C01818=1037.554,349.984,372.996,172.475,44.077,158.586
C01819=1037.561,350.231,372.958,172.480,44.080,158.587
C01820=1037.569,350.478,372.921,172.487,44.083,158.588
C01821=1037.577,350.725,372.883,172.492,44.085,158.589
C01822=1037.584,350.973,372.845,172.498,44.089,158.591
C01823=1037.592,351.220,372.808,172.503,44.092,158.592
C01824=1037.599,351.466,372.769,172.510,44.094,158.593
C01825=1037.607,351.714,372.731,172.515,44.097,158.594
C01826=1037.615,351.960,372.694,172.521,44.100,158.595
C01827=1037.623,352.207,372.656,172.526,44.102,158.596
C01828=1037.631,352.455,372.618,172.533,44.105,158.598
C01829=1037.638,352.702,372.580,172.538,44.108,158.599
C01830=1037.645,352.948,372.542,172.544,44.111,158.600
C01831=1037.653,353.196,372.504,172.550,44.114,158.601
C01832=1037.661,353.443,372.466,172.556,44.116,158.602
C01833=1037.668,353.689,372.427,172.561,44.119,158.604
C01834=1037.677,353.937,372.390,172.568,44.122,158.605
C01835=1037.685,354.183,372.352,172.574,44.125,158.606
C01836=1037.692,354.431,372.314,172.579,44.128,158.607
C01837=1037.700,354.678,372.276,172.586,44.130,158.608
C01838=1037.708,354.924,372.238,172.591,44.134,158.610
C01839=1037.716,355.171,372.199,172.598,44.136,158.611
C01840=1037.723,355.418,372.161,172.603,44.139,158.612
C01841=1037.731,355.666,372.123,172.609,44.142,158.613
C01842=1037.739,355.912,372.085,172.616,44.145,158.615
C01843=1037.747,356.159,372.047,172.621,44.148,158.616
C01844=1037.754,356.406,372.008,172.628,44.151,158.617
C01845=1037.762,356.653,371.969,172.633,44.154,158.619
C01846=1037.770,356.900,371.931,172.639,44.157,158.620
C01847=1037.778,357.147,371.892,172.646,44.160,158.621
C01848=1037.786,357.393,371.854,172.651,44.163,158.622
C01849=1037.794,357.641,371.815,172.658,44.166,158.624
C01850=1037.801,357.887,371.777,172.663,44.168,158.625
C01851=1037.810,358.134,371.739,172.670,44.172,158.626
C01852=1037.818,358.381,371.700,172.676,44.175,158.627
C01853=1037.825,358.628,371.662,172.681,44.178,158.629
C01854=1037.833,358.875,371.623,172.688,44.181,158.630
C01855=1037.841,359.122,371.585,172.694,44.184,158.631
C01856=1037.848,359.369,371.546,172.700,44.187,158.632
C01857=1037.857,359.616,371.506,172.706,44.190,158.634
C01858=1037.864,359.862,371.468,172.713,44.193,158.635
C01859=1037.873,360.110,371.429,172.718,44.196,158.636
C01860=1037.881,360.356,371.390,172.725,44.199,158.638
C01861=1037.889,360.603,371.352,172.731,44.202,158.639
C01862=1037.897,360.850,371.313,172.737,44.205,158.640
C01863=1037.904,361.097,371.273,172.744,44.208,158.642
C01864=1037.912,361.343,371.235,172.750,44.212,158.643
C01865=1037.920,361.591,371.196,172.757,44.215,158.644
C01866=1037.929,361.837,371.157,172.762,44.218,158.646
C01867=1037.937,362.084,371.119,172.769,44.221,158.647
C01868=1037.944,362.331,371.079,172.775,44.225,158.648
C01869=1037.952,362.578,371.040,172.782,44.228,158.650
C01870=1037.964,362.950,370.981,172.791,44.233,158.652
C01871=1037.975,363.322,370.922,172.801,44.237,158.654
C01872=1037.988,363.694,370.862,172.811,44.242,158.656
C01873=1037.999,364.067,370.803,172.819,44.248,158.658
C01874=1038.008,364.313,370.764,172.826,44.251,158.659
C01875=1038.016,364.560,370.724,172.833,44.254,158.661
C01876=1038.023,364.806,370.685,172.839,44.258,158.662
C01877=1038.031,365.053,370.645,172.846,44.261,158.664
C01878=1038.039,365.300,370.607,172.852,44.264,158.665
C01879=1038.048,365.547,370.567,172.858,44.267,158.666
C01880=1038.056,365.794,370.527,172.865,44.271,158.668
C01881=1038.064,366.040,370.488,172.872,44.274,158.669
C01882=1038.072,366.287,370.448,172.877,44.277,158.671
C01883=1038.080,366.534,370.409,172.884,44.281,158.672
C01884=1038.088,366.781,370.369,172.891,44.284,158.674
C01885=1038.096,367.027,370.330,172.897,44.288,158.675
C01886=1038.104,367.274,370.290,172.904,44.291,158.676
C01887=1038.113,367.521,370.250,172.911,44.295,158.678
C01888=1038.121,367.767,370.211,172.917,44.298,158.679
C01889=1038.129,368.014,370.171,172.924,44.302,158.681
C01890=1038.137,368.260,370.131,172.931,44.305,158.682
C01891=1038.145,368.507,370.091,172.938,44.308,158.684
C01892=1038.154,368.754,370.052,172.943,44.312,158.685
C01893=1038.161,369.001,370.012,172.950,44.315,158.687
C01894=1038.170,369.247,369.973,172.957,44.318,158.688
C01895=1038.178,369.493,369.932,172.964,44.322,158.690
C01896=1038.186,369.740,369.893,172.971,44.326,158.691
C01897=1038.195,369.988,369.852,172.977,44.329,158.692
C01898=1038.203,370.234,369.812,172.984,44.333,158.694
C01899=1038.211,370.480,369.772,172.991,44.336,158.696
C01900=1038.219,370.727,369.732,172.998,44.340,158.697
C01901=1038.228,370.973,369.692,173.005,44.343,158.699
C01902=1038.236,371.220,369.652,173.011,44.347,158.700
C01903=1038.243,371.467,369.612,173.018,44.351,158.702
C01904=1038.251,371.713,369.571,173.025,44.355,158.703
C01905=1038.260,371.960,369.530,173.032,44.358,158.705
C01906=1038.268,372.206,369.491,173.039,44.362,158.706
C01907=1038.276,372.453,369.450,173.046,44.366,158.708
C01908=1038.285,372.699,369.410,173.053,44.369,158.709
C01909=1038.293,372.947,369.369,173.059,44.373,158.711
C01910=1038.302,373.193,369.329,173.066,44.377,158.712
C01911=1038.310,373.439,369.289,173.073,44.380,158.714
C01912=1038.318,373.685,369.248,173.080,44.384,158.716
C01913=1038.326,373.932,369.207,173.087,44.388,158.717
C01914=1038.334,374.179,369.167,173.094,44.391,158.719
C01915=1038.343,374.425,369.127,173.101,44.395,158.720
C01916=1038.351,374.672,369.086,173.108,44.399,158.722
C01917=1038.359,374.918,369.045,173.115,44.403,158.724
C01918=1038.367,375.165,369.005,173.122,44.406,158.725
C01919=1038.376,375.412,368.964,173.130,44.411,158.727
C01920=1038.384,375.658,368.923,173.137,44.414,158.728
C01921=1038.393,375.904,368.883,173.144,44.418,158.730
C01922=1038.401,376.151,368.842,173.151,44.422,158.732
C01923=1038.410,376.397,368.801,173.158,44.426,158.733
C01924=1038.418,376.643,368.760,173.165,44.429,158.735
C01925=1038.426,376.890,368.719,173.172,44.433,158.736
C01926=1038.441,377.283,368.654,173.184,44.439,158.739
C01927=1038.454,377.675,368.590,173.195,44.446,158.742
C01928=1038.468,378.068,368.524,173.207,44.452,158.744
C01929=1038.482,378.461,368.459,173.218,44.458,158.747
C01930=1038.489,378.707,368.417,173.225,44.462,158.749
C01931=1038.498,378.954,368.376,173.233,44.467,158.750
C01932=1038.506,379.200,368.335,173.240,44.470,158.752
C01933=1038.515,379.447,368.294,173.247,44.474,158.754
C01934=1038.523,379.692,368.252,173.254,44.478,158.755
C01935=1038.532,379.939,368.211,173.261,44.483,158.757
C01936=1038.541,380.184,368.169,173.270,44.487,158.759
C01937=1038.549,380.431,368.128,173.277,44.491,158.761
C01938=1038.558,380.677,368.087,173.284,44.495,158.762
C01939=1038.566,380.923,368.045,173.292,44.499,158.764
C01940=1038.574,381.169,368.003,173.299,44.503,158.766
C01941=1038.583,381.416,367.962,173.306,44.507,158.768
C01942=1038.591,381.662,367.921,173.315,44.511,158.769
C01943=1038.600,381.908,367.879,173.322,44.516,158.771
C01944=1038.609,382.155,367.838,173.329,44.520,158.773
C01945=1038.618,382.401,367.796,173.336,44.524,158.775
C01946=1038.625,382.647,367.754,173.344,44.528,158.776
C01947=1038.634,382.893,367.712,173.352,44.532,158.778
C01948=1038.643,383.140,367.670,173.360,44.537,158.780
C01949=1038.652,383.386,367.629,173.367,44.541,158.782
C01950=1038.661,383.633,367.587,173.374,44.545,158.783
C01951=1038.669,383.878,367.546,173.383,44.549,158.785
C01952=1038.678,384.125,367.503,173.390,44.554,158.787
C01953=1038.687,384.371,367.462,173.397,44.558,158.789
C01954=1038.696,384.618,367.420,173.406,44.562,158.791
C01955=1038.704,384.864,367.378,173.413,44.567,158.793
C01956=1038.714,385.110,367.336,173.421,44.571,158.794
C01957=1038.722,385.356,367.293,173.428,44.575,158.796
C01958=1038.731,385.603,367.252,173.436,44.579,158.798
C01959=1038.740,385.849,367.210,173.444,44.584,158.800
C01960=1038.749,386.095,367.168,173.452,44.588,158.802
C01961=1038.758,386.341,367.126,173.460,44.593,158.804
C01962=1038.766,386.588,367.084,173.467,44.597,158.805
C01963=1038.775,386.834,367.041,173.476,44.601,158.807
C01964=1038.784,387.080,366.999,173.483,44.606,158.809
C01965=1038.794,387.326,366.957,173.492,44.610,158.811
C01966=1038.802,387.572,366.915,173.499,44.615,158.813
C01967=1038.811,387.818,366.872,173.508,44.619,158.815
C01968=1038.820,388.065,366.831,173.515,44.624,158.817
C01969=1038.829,388.311,366.787,173.523,44.628,158.819
C01970=1038.838,388.557,366.745,173.531,44.632,158.821
C01971=1038.847,388.803,366.703,173.539,44.637,158.823
C01972=1038.856,389.050,366.660,173.548,44.642,158.825
C01973=1038.865,389.295,366.618,173.555,44.646,158.826
C01974=1038.873,389.541,366.574,173.564,44.651,158.828
C01975=1038.883,389.787,366.532,173.571,44.655,158.830
C01976=1038.892,390.034,366.489,173.580,44.660,158.832
C01977=1038.901,390.280,366.447,173.588,44.665,158.834
C01978=1038.909,390.526,366.404,173.596,44.670,158.836
C01979=1038.918,390.772,366.361,173.604,44.674,158.838
C01980=1038.928,391.019,366.318,173.613,44.679,158.840
C01981=1038.937,391.264,366.276,173.621,44.684,158.842
C01982=1038.945,391.477,366.238,173.627,44.687,158.844
C01983=1038.952,391.691,366.201,173.635,44.692,158.846
C01984=1038.959,391.904,366.163,173.642,44.696,158.847
C01985=1038.967,392.117,366.126,173.649,44.700,158.849
C01986=1038.976,392.331,366.088,173.657,44.704,158.851
C01987=1038.983,392.544,366.051,173.664,44.709,158.853
C01988=1038.991,392.757,366.014,173.672,44.713,158.855
C01989=1038.999,392.971,365.976,173.679,44.717,158.856
C01990=1039.009,393.217,365.933,173.687,44.721,158.858
C01991=1039.017,393.463,365.890,173.696,44.726,158.861
C01992=1039.026,393.709,365.846,173.704,44.731,158.863
C01993=1039.036,393.955,365.804,173.712,44.736,158.865
C01994=1039.045,394.201,365.760,173.721,44.741,158.867
C01995=1039.054,394.447,365.717,173.730,44.746,158.869
C01996=1039.064,394.693,365.673,173.737,44.751,158.871
C01997=1039.072,394.939,365.630,173.746,44.756,158.873
C01998=1039.082,395.185,365.586,173.755,44.761,158.875
C01999=1039.091,395.430,365.543,173.764,44.766,158.877
C02000=1039.100,395.677,365.499,173.772,44.771,158.879
C02001=1039.109,395.922,365.456,173.781,44.776,158.882
C02002=1039.119,396.168,365.412,173.790,44.781,158.884
C02003=1039.127,396.414,365.368,173.799,44.786,158.886
C02004=1039.136,396.660,365.324,173.807,44.791,158.888
C02005=1039.147,396.906,365.281,173.815,44.796,158.890
C02006=1039.155,397.152,365.237,173.824,44.801,158.892
C02007=1039.165,397.398,365.193,173.833,44.806,158.895
C02008=1039.174,397.644,365.149,173.842,44.811,158.897
C02009=1039.183,397.889,365.105,173.851,44.816,158.899
C02010=1039.192,398.136,365.061,173.860,44.821,158.901
C02011=1039.203,398.381,365.018,173.869,44.826,158.903
C02012=1039.212,398.627,364.973,173.878,44.832,158.906
C02013=1039.221,398.873,364.930,173.887,44.837,158.908
C02014=1039.231,399.118,364.885,173.896,44.842,158.910
C02015=1039.240,399.365,364.841,173.904,44.848,158.912
C02016=1039.249,399.611,364.797,173.913,44.853,158.914
C02017=1039.259,399.857,364.753,173.922,44.858,158.917
C02018=1039.268,400.102,364.708,173.931,44.863,158.919
C02019=1039.277,400.348,364.664,173.940,44.868,158.921
C02020=1039.287,400.594,364.620,173.949,44.874,158.924
C02021=1039.296,400.839,364.575,173.958,44.879,158.926
C02022=1039.306,401.086,364.531,173.968,44.884,158.928
C02023=1039.316,401.331,364.486,173.978,44.890,158.931
C02024=1039.325,401.577,364.442,173.987,44.895,158.933
C02025=1039.335,401.823,364.397,173.996,44.901,158.935
C02026=1039.344,402.068,364.352,174.005,44.906,158.938
C02027=1039.354,402.314,364.308,174.014,44.911,158.940
C02028=1039.363,402.560,364.263,174.023,44.917,158.942
C02029=1039.373,402.805,364.219,174.032,44.922,158.945
C02030=1039.382,403.051,364.173,174.042,44.928,158.947
C02031=1039.392,403.298,364.129,174.051,44.934,158.949
C02032=1039.402,403.544,364.084,174.061,44.939,158.952
C02033=1039.412,403.789,364.039,174.070,44.944,158.954
C02034=1039.421,404.035,363.994,174.080,44.950,158.957
C02035=1039.430,404.280,363.949,174.089,44.956,158.959
C02036=1039.440,404.526,363.904,174.098,44.961,158.961
C02037=1039.450,404.771,363.859,174.108,44.967,158.964
C02038=1039.459,405.018,363.813,174.118,44.973,158.966
C02039=1039.469,405.263,363.768,174.127,44.978,158.969
C02040=1039.479,405.508,363.723,174.137,44.984,158.971
C02041=1039.488,405.754,363.678,174.147,44.989,158.974
C02042=1039.498,405.978,363.637,174.155,44.995,158.976
C02043=1039.506,406.201,363.595,174.164,45.000,158.978
C02044=1039.515,406.424,363.554,174.173,45.005,158.981
C02045=1039.525,406.647,363.513,174.182,45.010,158.983
C02046=1039.533,406.870,363.471,174.190,45.016,158.985
C02047=1039.542,407.093,363.431,174.199,45.021,158.987
C02048=1039.551,407.317,363.389,174.208,45.026,158.990
C02049=1039.560,407.540,363.347,174.218,45.032,158.992
C02050=1039.570,407.786,363.302,174.227,45.038,158.995
C02051=1039.580,408.031,363.256,174.238,45.043,158.997
C02052=1039.590,408.277,363.211,174.247,45.049,159.000
C02053=1039.599,408.523,363.165,174.257,45.055,159.002
C02054=1039.609,408.769,363.120,174.267,45.061,159.005
C02055=1039.620,409.014,363.074,174.277,45.067,159.007
C02056=1039.629,409.260,363.028,174.287,45.073,159.010
C02057=1039.640,409.505,362.982,174.297,45.079,159.013
C02058=1039.650,409.750,362.936,174.307,45.084,159.015
C02059=1039.660,409.997,362.890,174.318,45.090,159.018
C02060=1039.670,410.242,362.844,174.327,45.097,159.020
C02061=1039.680,410.487,362.799,174.338,45.102,159.023
C02062=1039.690,410.733,362.752,174.348,45.109,159.026
C02063=1039.701,410.979,362.706,174.358,45.115,159.028
C02064=1039.711,411.223,362.661,174.369,45.120,159.031
C02065=1039.721,411.469,362.614,174.379,45.127,159.034
C02066=1039.731,411.715,362.569,174.389,45.133,159.037
C02067=1039.741,411.960,362.521,174.400,45.139,159.039
C02068=1039.751,412.206,362.475,174.410,45.145,159.042
C02069=1039.762,412.452,362.429,174.420,45.152,159.045
C02070=1039.772,412.696,362.382,174.431,45.158,159.047
C02071=1039.781,412.942,362.336,174.441,45.164,159.050
C02072=1039.792,413.188,362.290,174.452,45.170,159.053
C02073=1039.802,413.433,362.242,174.462,45.176,159.056
C02074=1039.812,413.679,362.196,174.473,45.183,159.058
C02075=1039.823,413.924,362.149,174.484,45.189,159.061
C02076=1039.833,414.169,362.102,174.494,45.196,159.064
C02077=1039.843,414.415,362.056,174.505,45.202,159.067
C02078=1039.854,414.660,362.009,174.516,45.208,159.070
C02079=1039.864,414.905,361.962,174.527,45.215,159.073
C02080=1039.874,415.151,361.915,174.538,45.221,159.075
C02081=1039.884,415.397,361.868,174.548,45.228,159.078
C02082=1039.895,415.642,361.821,174.559,45.234,159.081
C02083=1039.905,415.887,361.774,174.570,45.241,159.084
C02084=1039.916,416.132,361.727,174.581,45.247,159.087
C02085=1039.927,416.378,361.680,174.592,45.254,159.090
C02086=1039.937,416.623,361.633,174.603,45.260,159.093
C02087=1039.948,416.868,361.586,174.614,45.266,159.096
C02088=1039.959,417.113,361.539,174.625,45.273,159.099
C02089=1039.969,417.359,361.492,174.636,45.280,159.102
C02090=1039.980,417.605,361.444,174.647,45.286,159.104
C02091=1039.990,417.850,361.397,174.658,45.293,159.107
C02092=1040.001,418.095,361.349,174.670,45.300,159.110
C02093=1040.011,418.341,361.301,174.681,45.306,159.113
C02094=1040.021,418.585,361.253,174.692,45.313,159.116
C02095=1040.032,418.831,361.206,174.704,45.320,159.119
C02096=1040.043,419.076,361.158,174.715,45.327,159.123
C02097=1040.053,419.321,361.111,174.726,45.334,159.126
C02098=1040.064,419.566,361.062,174.738,45.340,159.129
C02099=1040.075,419.811,361.016,174.749,45.347,159.132
C02100=1040.086,420.057,360.968,174.761,45.354,159.135
C02101=1040.097,420.301,360.920,174.772,45.361,159.138
C02102=1040.106,420.529,360.875,174.783,45.367,159.141
C02103=1040.116,420.756,360.831,174.793,45.374,159.144
C02104=1040.126,420.985,360.786,174.804,45.380,159.146
C02105=1040.136,421.211,360.741,174.815,45.387,159.149
C02106=1040.146,421.439,360.697,174.826,45.393,159.152
C02107=1040.156,421.666,360.652,174.837,45.399,159.155
C02108=1040.167,421.894,360.607,174.848,45.406,159.158
C02109=1040.176,422.121,360.563,174.859,45.412,159.161
C02110=1040.187,422.367,360.514,174.871,45.419,159.164
C02111=1040.198,422.611,360.466,174.883,45.426,159.168
C02112=1040.209,422.856,360.417,174.895,45.434,159.171
C02113=1040.220,423.101,360.369,174.907,45.440,159.174
C02114=1040.232,423.347,360.321,174.919,45.448,159.177
C02115=1040.243,423.592,360.272,174.931,45.455,159.181
C02116=1040.253,423.836,360.224,174.943,45.462,159.184
C02117=1040.265,424.082,360.176,174.955,45.469,159.187
C02118=1040.276,424.326,360.127,174.968,45.476,159.190
C02119=1040.287,424.572,360.078,174.979,45.484,159.194
C02120=1040.298,424.816,360.029,174.992,45.491,159.197
C02121=1040.309,425.061,359.980,175.005,45.498,159.200
C02122=1040.320,425.307,359.931,175.016,45.506,159.204
C02123=1040.332,425.552,359.882,175.029,45.513,159.207
C02124=1040.343,425.796,359.833,175.042,45.520,159.211
C02125=1040.354,426.041,359.784,175.054,45.528,159.214
C02126=1040.365,426.286,359.735,175.066,45.535,159.217
C02127=1040.377,426.531,359.686,175.079,45.543,159.221
C02128=1040.388,426.776,359.637,175.092,45.550,159.224
C02129=1040.399,427.021,359.587,175.104,45.557,159.228
C02130=1040.410,427.265,359.538,175.117,45.565,159.231
C02131=1040.421,427.510,359.489,175.130,45.572,159.234
C02132=1040.433,427.756,359.440,175.143,45.580,159.238
C02133=1040.444,428.001,359.390,175.156,45.588,159.242
C02134=1040.456,428.245,359.340,175.168,45.595,159.245
C02135=1040.467,428.490,359.291,175.182,45.603,159.249
C02136=1040.478,428.735,359.241,175.194,45.610,159.252
C02137=1040.490,428.979,359.192,175.207,45.618,159.256
C02138=1040.501,429.224,359.142,175.220,45.626,159.259
C02139=1040.513,429.469,359.092,175.233,45.634,159.263
C02140=1040.524,429.714,359.042,175.246,45.642,159.267
C02141=1040.536,429.958,358.993,175.260,45.649,159.270
C02142=1040.547,430.204,358.942,175.273,45.657,159.274
C02143=1040.559,430.448,358.892,175.286,45.665,159.278
C02144=1040.570,430.692,358.842,175.300,45.673,159.281
C02145=1040.582,430.937,358.792,175.313,45.681,159.285
C02146=1040.593,431.181,358.741,175.326,45.689,159.289
C02147=1040.605,431.426,358.691,175.339,45.697,159.292
C02148=1040.617,431.671,358.641,175.353,45.704,159.296
C02149=1040.629,431.915,358.591,175.367,45.713,159.300
C02150=1040.640,432.161,358.540,175.380,45.720,159.303
C02151=1040.652,432.405,358.490,175.394,45.728,159.307
C02152=1040.664,432.649,358.439,175.407,45.736,159.311
C02153=1040.676,432.894,358.389,175.422,45.745,159.315
C02154=1040.688,433.139,358.338,175.435,45.752,159.319
C02155=1040.700,433.383,358.288,175.449,45.761,159.322
C02156=1040.711,433.628,358.237,175.463,45.769,159.326
C02157=1040.724,433.872,358.186,175.477,45.777,159.330
C02158=1040.736,434.117,358.136,175.491,45.785,159.334
C02159=1040.748,434.361,358.085,175.505,45.794,159.338
C02160=1040.760,434.606,358.034,175.520,45.802,159.342
C02161=1040.772,434.850,357.984,175.533,45.810,159.346
C02162=1040.783,435.085,357.935,175.547,45.817,159.350
C02163=1040.795,435.319,357.885,175.561,45.826,159.353
C02164=1040.807,435.554,357.836,175.574,45.834,159.357
C02165=1040.818,435.788,357.787,175.588,45.842,159.361
C02166=1040.829,436.022,357.738,175.602,45.850,159.365
C02167=1040.842,436.256,357.689,175.616,45.858,159.369
C02168=1040.853,436.491,357.639,175.630,45.866,159.373
C02169=1040.865,436.726,357.591,175.644,45.874,159.377
C02170=1040.877,436.969,357.538,175.659,45.882,159.381
C02171=1040.889,437.214,357.487,175.674,45.891,159.385
C02172=1040.901,437.458,357.436,175.688,45.899,159.389
C02173=1040.914,437.702,357.384,175.703,45.908,159.393
C02174=1040.926,437.947,357.332,175.718,45.917,159.397
C02175=1040.939,438.191,357.280,175.733,45.925,159.401
C02176=1040.951,438.436,357.229,175.748,45.934,159.406
C02177=1040.963,438.680,357.177,175.763,45.943,159.410
C02178=1040.976,438.924,357.124,175.777,45.951,159.414
C02179=1040.988,439.168,357.073,175.793,45.960,159.418
C02180=1041.001,439.412,357.020,175.808,45.969,159.423
C02181=1041.013,439.657,356.969,175.823,45.978,159.427
C02182=1041.026,439.901,356.916,175.839,45.987,159.431
C02183=1041.038,440.145,356.864,175.854,45.996,159.435
C02184=1041.051,440.390,356.812,175.869,46.005,159.440
C02185=1041.063,440.633,356.759,175.885,46.013,159.444
C02186=1041.076,440.878,356.706,175.900,46.022,159.448
C02187=1041.088,441.122,356.654,175.916,46.031,159.453
C02188=1041.101,441.366,356.602,175.931,46.040,159.457
C02189=1041.114,441.610,356.549,175.948,46.049,159.462
C02190=1041.126,441.854,356.496,175.963,46.058,159.466
C02191=1041.140,442.098,356.443,175.979,46.067,159.470
C02192=1041.153,442.342,356.391,175.995,46.076,159.475
C02193=1041.166,442.586,356.338,176.011,46.086,159.480
C02194=1041.179,442.830,356.285,176.026,46.095,159.484
C02195=1041.191,443.074,356.233,176.043,46.104,159.489
C02196=1041.205,443.318,356.180,176.059,46.113,159.493
C02197=1041.218,443.562,356.126,176.076,46.122,159.498
C02198=1041.231,443.806,356.073,176.091,46.131,159.502
C02199=1041.244,444.050,356.020,176.108,46.141,159.507
C02200=1041.257,444.294,355.967,176.124,46.150,159.512
C02201=1041.270,444.538,355.914,176.141,46.159,159.516
C02202=1041.283,444.781,355.860,176.157,46.169,159.521
C02203=1041.296,445.023,355.807,176.174,46.178,159.526
C02204=1041.311,445.266,355.755,176.191,46.187,159.530
C02205=1041.326,445.511,355.703,176.207,46.196,159.535
C02206=1041.341,445.754,355.652,176.224,46.206,159.540
C02207=1041.356,445.997,355.601,176.241,46.214,159.544
C02208=1041.374,446.241,355.550,176.258,46.223,159.549
C02209=1041.390,446.485,355.500,176.275,46.232,159.553
C02210=1041.408,446.729,355.451,176.292,46.240,159.558
C02211=1041.427,446.973,355.401,176.309,46.248,159.562
C02212=1041.446,447.217,355.353,176.327,46.257,159.567
C02213=1041.465,447.462,355.305,176.344,46.265,159.571
C02214=1041.485,447.706,355.257,176.361,46.273,159.576
C02215=1041.506,447.950,355.210,176.380,46.281,159.580
C02216=1041.527,448.195,355.163,176.397,46.289,159.585
C02217=1041.549,448.440,355.116,176.415,46.296,159.589
C02218=1041.571,448.684,355.070,176.432,46.305,159.594
C02219=1041.595,448.929,355.025,176.450,46.312,159.598
C02220=1041.619,449.175,354.981,176.468,46.320,159.602
C02221=1041.643,449.419,354.936,176.486,46.327,159.607
C02222=1041.671,449.706,354.885,176.507,46.335,159.612
C02223=1041.702,449.993,354.834,176.529,46.344,159.617
C02224=1041.732,450.280,354.784,176.550,46.352,159.622
C02225=1041.764,450.567,354.735,176.571,46.360,159.627
C02226=1041.791,450.813,354.693,176.590,46.367,159.631
C02227=1041.820,451.059,354.652,176.608,46.373,159.635
C02228=1041.849,451.304,354.611,176.627,46.380,159.639
C02229=1041.878,451.549,354.571,176.645,46.387,159.644
C02230=1041.579,451.594,354.255,176.648,46.464,159.667
C02231=1041.550,451.349,354.295,176.629,46.458,159.663
C02232=1041.521,451.104,354.336,176.611,46.452,159.659
C02233=1041.493,450.858,354.377,176.592,46.445,159.655
C02234=1041.465,450.612,354.419,176.573,46.438,159.650
C02235=1041.435,450.341,354.465,176.553,46.431,159.646
C02236=1041.405,450.068,354.512,176.533,46.423,159.641
C02237=1041.376,449.797,354.560,176.513,46.415,159.636
C02238=1041.349,449.525,354.608,176.492,46.407,159.631
C02239=1041.324,449.280,354.652,176.474,46.400,159.627
C02240=1041.300,449.035,354.698,176.456,46.392,159.623
C02241=1041.276,448.790,354.742,176.438,46.385,159.618
C02242=1041.254,448.546,354.787,176.420,46.378,159.614
C02243=1041.231,448.301,354.834,176.403,46.370,159.609
C02244=1041.210,448.056,354.880,176.385,46.362,159.605
C02245=1041.189,447.812,354.928,176.368,46.354,159.601
C02246=1041.169,447.568,354.975,176.349,46.346,159.596
C02247=1041.148,447.323,355.023,176.332,46.338,159.592
C02248=1041.130,447.079,355.071,176.315,46.330,159.587
C02249=1041.111,446.834,355.120,176.298,46.322,159.583
C02250=1041.093,446.591,355.169,176.280,46.313,159.578
C02251=1041.075,446.346,355.219,176.263,46.305,159.574
C02252=1041.058,446.103,355.269,176.246,46.296,159.569
C02253=1041.041,445.859,355.320,176.229,46.288,159.564
C02254=1041.026,445.616,355.371,176.213,46.279,159.560
C02255=1041.011,445.372,355.423,176.195,46.270,159.555
C02256=1040.996,445.128,355.475,176.178,46.261,159.551
C02257=1040.983,444.886,355.527,176.162,46.252,159.546
C02258=1040.969,444.642,355.580,176.145,46.243,159.541
C02259=1040.956,444.399,355.634,176.129,46.233,159.537
C02260=1040.942,444.155,355.687,176.112,46.224,159.532
C02261=1040.929,443.911,355.740,176.095,46.215,159.527
C02262=1040.916,443.667,355.793,176.079,46.206,159.523
C02263=1040.903,443.423,355.846,176.063,46.196,159.518
C02264=1040.891,443.179,355.899,176.047,46.187,159.514
C02265=1040.878,442.935,355.953,176.031,46.178,159.509
C02266=1040.864,442.691,356.006,176.014,46.169,159.504
C02267=1040.852,442.447,356.058,175.999,46.160,159.500
C02268=1040.839,442.203,356.111,175.982,46.151,159.495
C02269=1040.826,441.960,356.164,175.966,46.142,159.491
C02270=1040.813,441.715,356.217,175.951,46.133,159.486
C02271=1040.800,441.471,356.270,175.935,46.124,159.482
C02272=1040.787,441.226,356.322,175.919,46.115,159.478
C02273=1040.774,440.983,356.374,175.903,46.107,159.473
C02274=1040.761,440.739,356.427,175.888,46.098,159.469
C02275=1040.749,440.495,356.479,175.872,46.089,159.464
C02276=1040.736,440.250,356.532,175.857,46.080,159.460
C02277=1040.724,440.006,356.584,175.842,46.071,159.456
C02278=1040.711,439.762,356.636,175.825,46.062,159.451
C02279=1040.699,439.517,356.689,175.811,46.054,159.447
C02280=1040.686,439.273,356.741,175.795,46.045,159.443
C02281=1040.674,439.030,356.792,175.780,46.036,159.439
C02282=1040.661,438.785,356.845,175.764,46.027,159.434
C02283=1040.649,438.541,356.896,175.750,46.019,159.430
C02284=1040.637,438.297,356.949,175.735,46.010,159.426
C02285=1040.624,438.052,357.001,175.720,46.002,159.422
C02286=1040.612,437.808,357.052,175.705,45.993,159.418
C02287=1040.599,437.564,357.104,175.690,45.985,159.414
C02288=1040.587,437.320,357.155,175.675,45.976,159.409
C02289=1040.575,437.074,357.207,175.661,45.968,159.405
C02290=1040.563,436.831,357.259,175.646,45.959,159.401
C02291=1040.551,436.596,357.308,175.631,45.951,159.397
C02292=1040.538,436.361,357.358,175.618,45.943,159.393
C02293=1040.527,436.126,357.407,175.603,45.935,159.389
C02294=1040.515,435.891,357.457,175.590,45.927,159.386
C02295=1040.504,435.656,357.506,175.575,45.919,159.382
C02296=1040.492,435.420,357.555,175.562,45.911,159.378
C02297=1040.480,435.185,357.605,175.548,45.903,159.374
C02298=1040.469,434.950,357.653,175.534,45.895,159.370
C02299=1040.456,434.706,357.704,175.520,45.887,159.366
C02300=1040.445,434.461,357.755,175.505,45.879,159.362
C02301=1040.432,434.217,357.806,175.492,45.870,159.358
C02302=1040.420,433.972,357.857,175.478,45.863,159.355
C02303=1040.408,433.728,357.907,175.463,45.855,159.351
C02304=1040.397,433.484,357.958,175.450,45.846,159.347
C02305=1040.384,433.239,358.008,175.435,45.838,159.343
C02306=1040.372,432.994,358.060,175.422,45.830,159.339
C02307=1040.360,432.749,358.110,175.407,45.822,159.335
C02308=1040.349,432.505,358.160,175.394,45.815,159.332
C02309=1040.337,432.260,358.210,175.380,45.806,159.328
C02310=1040.325,432.016,358.262,175.367,45.799,159.324
C02311=1040.313,431.772,358.311,175.353,45.791,159.320
C02312=1040.302,431.526,358.362,175.339,45.783,159.317
C02313=1040.290,431.282,358.412,175.326,45.775,159.313
C02314=1040.278,431.037,358.463,175.312,45.767,159.309
C02315=1040.266,430.792,358.513,175.299,45.759,159.305
C02316=1040.255,430.548,358.563,175.285,45.751,159.302
C02317=1040.243,430.304,358.613,175.272,45.743,159.298
C02318=1040.232,430.058,358.663,175.258,45.736,159.294
C02319=1040.220,429.814,358.712,175.245,45.728,159.291
C02320=1040.209,429.569,358.763,175.232,45.721,159.287
C02321=1040.197,429.325,358.813,175.219,45.713,159.283
C02322=1040.186,429.080,358.862,175.206,45.705,159.280
C02323=1040.174,428.835,358.913,175.193,45.697,159.276
C02324=1040.163,428.590,358.962,175.180,45.690,159.273
C02325=1040.152,428.346,359.012,175.167,45.683,159.269
C02326=1040.141,428.101,359.062,175.153,45.675,159.266
C02327=1040.129,427.855,359.111,175.141,45.667,159.262
C02328=1040.117,427.611,359.161,175.128,45.660,159.259
C02329=1040.106,427.366,359.210,175.115,45.653,159.255
C02330=1040.095,427.121,359.259,175.103,45.645,159.252
C02331=1040.084,426.877,359.308,175.090,45.638,159.248
C02332=1040.072,426.631,359.358,175.077,45.630,159.245
C02333=1040.060,426.386,359.407,175.065,45.623,159.241
C02334=1040.049,426.142,359.456,175.052,45.615,159.238
C02335=1040.038,425.897,359.505,175.039,45.608,159.235
C02336=1040.027,425.652,359.554,175.027,45.601,159.231
C02337=1040.016,425.407,359.603,175.015,45.593,159.228
C02338=1040.004,425.162,359.652,175.002,45.586,159.225
C02339=1039.994,424.917,359.701,174.989,45.579,159.221
C02340=1039.982,424.672,359.750,174.977,45.572,159.218
C02341=1039.971,424.427,359.799,174.965,45.564,159.214
C02342=1039.960,424.182,359.847,174.953,45.557,159.211
C02343=1039.949,423.937,359.895,174.940,45.550,159.208
C02344=1039.938,423.692,359.944,174.929,45.543,159.205
C02345=1039.927,423.447,359.993,174.916,45.536,159.201
C02346=1039.916,423.201,360.042,174.905,45.529,159.198
C02347=1039.904,422.957,360.090,174.892,45.522,159.195
C02348=1039.893,422.712,360.138,174.880,45.515,159.192
C02349=1039.883,422.467,360.186,174.868,45.508,159.188
C02350=1039.872,422.222,360.235,174.856,45.501,159.185
C02351=1039.862,421.993,360.280,174.845,45.494,159.182
C02352=1039.851,421.764,360.325,174.834,45.488,159.179
C02353=1039.841,421.536,360.370,174.822,45.482,159.176
C02354=1039.831,421.307,360.415,174.812,45.475,159.173
C02355=1039.821,421.079,360.460,174.801,45.469,159.170
C02356=1039.811,420.850,360.504,174.790,45.462,159.167
C02357=1039.801,420.622,360.549,174.779,45.456,159.165
C02358=1039.791,420.394,360.594,174.768,45.450,159.162
C02359=1039.780,420.148,360.642,174.757,45.443,159.159
C02360=1039.770,419.903,360.689,174.745,45.436,159.155
C02361=1039.758,419.658,360.738,174.734,45.429,159.152
C02362=1039.748,419.413,360.786,174.722,45.422,159.149
C02363=1039.737,419.167,360.833,174.711,45.415,159.146
C02364=1039.727,418.923,360.881,174.699,45.409,159.143
C02365=1039.716,418.677,360.928,174.688,45.402,159.140
C02366=1039.705,418.432,360.977,174.677,45.396,159.137
C02367=1039.695,418.187,361.024,174.665,45.389,159.134
C02368=1039.685,417.942,361.072,174.654,45.382,159.131
C02369=1039.674,417.696,361.119,174.642,45.376,159.128
C02370=1039.663,417.451,361.166,174.631,45.369,159.125
C02371=1039.653,417.206,361.213,174.620,45.363,159.122
C02372=1039.642,416.960,361.261,174.609,45.356,159.119
C02373=1039.632,416.714,361.308,174.598,45.350,159.116
C02374=1039.621,416.469,361.355,174.587,45.343,159.113
C02375=1039.611,416.224,361.402,174.576,45.337,159.111
C02376=1039.600,415.978,361.449,174.565,45.330,159.108
C02377=1039.589,415.733,361.496,174.554,45.324,159.105
C02378=1039.579,415.488,361.543,174.543,45.318,159.102
C02379=1039.569,415.243,361.590,174.532,45.311,159.099
C02380=1039.558,414.998,361.637,174.521,45.305,159.096
C02381=1039.547,414.752,361.684,174.510,45.299,159.093
C02382=1039.538,414.506,361.731,174.500,45.292,159.091
C02383=1039.527,414.261,361.777,174.489,45.286,159.088
C02384=1039.516,414.016,361.825,174.478,45.279,159.085
C02385=1039.507,413.770,361.871,174.468,45.273,159.082
C02386=1039.496,413.525,361.918,174.457,45.267,159.079
C02387=1039.486,413.279,361.964,174.446,45.261,159.077
C02388=1039.476,413.034,362.011,174.436,45.255,159.074
C02389=1039.465,412.789,362.057,174.425,45.248,159.071
C02390=1039.455,412.543,362.105,174.415,45.242,159.068
C02391=1039.445,412.298,362.151,174.404,45.236,159.065
C02392=1039.435,412.052,362.197,174.394,45.230,159.063
C02393=1039.425,411.807,362.244,174.383,45.224,159.060
C02394=1039.415,411.561,362.290,174.373,45.217,159.057
C02395=1039.404,411.316,362.336,174.362,45.212,159.055
C02396=1039.394,411.071,362.382,174.352,45.206,159.052
C02397=1039.384,410.825,362.428,174.342,45.199,159.049
C02398=1039.374,410.579,362.474,174.331,45.194,159.047
C02399=1039.363,410.334,362.520,174.321,45.188,159.044
C02400=1039.354,410.088,362.566,174.311,45.181,159.041
C02401=1039.343,409.843,362.612,174.301,45.176,159.039
C02402=1039.333,409.597,362.659,174.291,45.170,159.036
C02403=1039.323,409.351,362.703,174.281,45.164,159.033
C02404=1039.313,409.106,362.749,174.271,45.158,159.031
C02405=1039.303,408.860,362.796,174.260,45.152,159.028
C02406=1039.293,408.615,362.841,174.250,45.147,159.026
C02407=1039.283,408.369,362.887,174.240,45.141,159.023
C02408=1039.273,408.124,362.933,174.230,45.135,159.021
C02409=1039.263,407.878,362.979,174.220,45.129,159.018
C02410=1039.253,407.633,363.023,174.211,45.123,159.015
C02411=1039.244,407.408,363.066,174.202,45.117,159.013
C02412=1039.235,407.184,363.107,174.193,45.113,159.011
C02413=1039.226,406.959,363.148,174.183,45.107,159.008
C02414=1039.217,406.735,363.190,174.174,45.102,159.006
C02415=1039.208,406.511,363.232,174.165,45.097,159.004
C02416=1039.199,406.286,363.272,174.156,45.092,159.002
C02417=1039.190,406.062,363.314,174.148,45.086,158.999
C02418=1039.181,405.838,363.356,174.139,45.082,158.997
C02419=1039.171,405.592,363.401,174.130,45.075,158.995
C02420=1039.162,405.346,363.446,174.119,45.070,158.992
C02421=1039.152,405.101,363.491,174.110,45.064,158.990
C02422=1039.142,404.855,363.536,174.101,45.059,158.987
C02423=1039.132,404.609,363.583,174.090,45.054,158.985
C02424=1039.123,404.364,363.627,174.081,45.048,158.982
C02425=1039.113,404.118,363.672,174.072,45.042,158.980
C02426=1039.104,403.873,363.718,174.062,45.037,158.978
C02427=1039.094,403.627,363.762,174.052,45.031,158.975
C02428=1039.085,403.381,363.807,174.043,45.026,158.973
C02429=1039.075,403.135,363.852,174.034,45.020,158.970
C02430=1039.065,402.889,363.897,174.025,45.015,158.968
C02431=1039.056,402.643,363.942,174.015,45.010,158.966
C02432=1039.046,402.398,363.987,174.006,45.004,158.963
C02433=1039.037,402.152,364.031,173.996,44.999,158.961
C02434=1039.027,401.906,364.076,173.987,44.993,158.959
C02435=1039.017,401.661,364.121,173.978,44.988,158.956
C02436=1039.008,401.415,364.165,173.968,44.982,158.954
C02437=1038.998,401.169,364.209,173.959,44.977,158.952
C02438=1038.989,400.923,364.254,173.950,44.972,158.949
C02439=1038.979,400.677,364.298,173.941,44.966,158.947
C02440=1038.970,400.431,364.343,173.932,44.962,158.945
C02441=1038.960,400.186,364.387,173.923,44.956,158.942
C02442=1038.951,399.940,364.431,173.914,44.951,158.940
C02443=1038.942,399.694,364.475,173.905,44.946,158.938
C02444=1038.932,399.449,364.520,173.896,44.941,158.936
C02445=1038.923,399.202,364.564,173.887,44.935,158.933
C02446=1038.913,398.956,364.608,173.878,44.930,158.931
C02447=1038.903,398.711,364.652,173.869,44.925,158.929
C02448=1038.894,398.465,364.695,173.860,44.920,158.927
C02449=1038.885,398.219,364.740,173.851,44.915,158.924
C02450=1038.875,397.973,364.784,173.842,44.910,158.922
C02451=1038.866,397.727,364.829,173.833,44.905,158.920
C02452=1038.857,397.482,364.872,173.824,44.900,158.918
C02453=1038.847,397.236,364.916,173.815,44.894,158.916
C02454=1038.837,396.990,364.960,173.806,44.889,158.913
C02455=1038.829,396.744,365.003,173.798,44.884,158.911
C02456=1038.819,396.498,365.047,173.789,44.879,158.909
C02457=1038.810,396.252,365.091,173.780,44.874,158.907
C02458=1038.801,396.006,365.135,173.771,44.869,158.905
C02459=1038.792,395.760,365.179,173.762,44.864,158.903
C02460=1038.783,395.514,365.221,173.754,44.860,158.901
C02461=1038.773,395.268,365.266,173.746,44.855,158.898
C02462=1038.764,395.023,365.309,173.737,44.850,158.896
C02463=1038.755,394.776,365.353,173.728,44.845,158.894
C02464=1038.746,394.531,365.396,173.719,44.840,158.892
C02465=1038.737,394.284,365.439,173.711,44.835,158.890
C02466=1038.727,394.039,365.482,173.703,44.830,158.888
C02467=1038.718,393.792,365.526,173.694,44.826,158.886
C02468=1038.709,393.547,365.569,173.685,44.821,158.884
C02469=1038.699,393.300,365.612,173.677,44.816,158.882
C02470=1038.690,393.055,365.656,173.669,44.811,158.880
C02471=1038.683,392.840,365.693,173.661,44.807,158.878
C02472=1038.675,392.626,365.731,173.654,44.803,158.876
C02473=1038.667,392.411,365.769,173.646,44.799,158.874
C02474=1038.659,392.197,365.807,173.639,44.795,158.873
C02475=1038.651,391.983,365.844,173.632,44.791,158.871
C02476=1038.643,391.768,365.881,173.624,44.787,158.869
C02477=1038.635,391.554,365.919,173.617,44.783,158.867
C02478=1038.628,391.339,365.957,173.610,44.778,158.865
C02479=1038.618,391.094,365.999,173.602,44.774,158.864
C02480=1038.610,390.848,366.042,173.593,44.769,158.862
C02481=1038.600,390.601,366.085,173.586,44.764,158.859
C02482=1038.591,390.355,366.128,173.577,44.760,158.857
C02483=1038.582,390.109,366.170,173.569,44.755,158.856
C02484=1038.574,389.863,366.213,173.561,44.750,158.854
C02485=1038.564,389.617,366.256,173.552,44.746,158.852
C02486=1038.556,389.370,366.299,173.545,44.741,158.850
C02487=1038.546,389.124,366.341,173.536,44.737,158.848
C02488=1038.538,388.878,366.384,173.528,44.732,158.846
C02489=1038.529,388.633,366.426,173.520,44.728,158.844
C02490=1038.520,388.387,366.469,173.512,44.724,158.842
C02491=1038.511,388.140,366.511,173.504,44.719,158.840
C02492=1038.502,387.894,366.554,173.496,44.714,158.838
C02493=1038.493,387.647,366.596,173.488,44.710,158.836
C02494=1038.484,387.401,366.639,173.480,44.706,158.834
C02495=1038.475,387.155,366.680,173.472,44.701,158.832
C02496=1038.466,386.909,366.723,173.464,44.697,158.830
C02497=1038.458,386.663,366.765,173.457,44.693,158.829
C02498=1038.448,386.417,366.808,173.448,44.688,158.827
C02499=1038.439,386.170,366.849,173.441,44.684,158.825
C02500=1038.431,385.924,366.891,173.432,44.680,158.823
C02501=1038.421,385.678,366.933,173.425,44.675,158.821
C02502=1038.413,385.432,366.976,173.417,44.671,158.819
C02503=1038.404,385.185,367.018,173.409,44.667,158.818
C02504=1038.395,384.940,367.060,173.402,44.663,158.816
C02505=1038.386,384.693,367.102,173.393,44.658,158.814
C02506=1038.377,384.447,367.143,173.386,44.654,158.812
C02507=1038.368,384.200,367.185,173.378,44.650,158.810
C02508=1038.360,383.954,367.227,173.370,44.645,158.808
C02509=1038.352,383.708,367.269,173.362,44.641,158.807
C02510=1038.343,383.462,367.310,173.355,44.637,158.805
C02511=1038.334,383.215,367.352,173.348,44.633,158.803
C02512=1038.325,382.969,367.394,173.339,44.629,158.801
C02513=1038.317,382.722,367.436,173.332,44.625,158.800
C02514=1038.308,382.477,367.478,173.325,44.621,158.798
C02515=1038.299,382.230,367.519,173.316,44.616,158.796
C02516=1038.290,381.984,367.561,173.309,44.612,158.794
C02517=1038.281,381.738,367.603,173.302,44.608,158.792
C02518=1038.273,381.492,367.644,173.294,44.604,158.791
C02519=1038.265,381.245,367.686,173.287,44.600,158.789
C02520=1038.256,380.998,367.727,173.279,44.596,158.787
C02521=1038.248,380.753,367.769,173.272,44.592,158.785
C02522=1038.239,380.506,367.810,173.264,44.588,158.784
C02523=1038.230,380.259,367.851,173.257,44.584,158.782
C02524=1038.222,380.014,367.893,173.250,44.580,158.780
C02525=1038.213,379.767,367.935,173.242,44.575,158.779
C02526=1038.205,379.520,367.976,173.234,44.571,158.777
C02527=1038.197,379.274,368.017,173.227,44.568,158.775
C02528=1038.188,379.027,368.058,173.220,44.564,158.773
C02529=1038.180,378.782,368.100,173.212,44.559,158.772
C02530=1038.171,378.535,368.141,173.205,44.556,158.770
C02531=1038.158,378.140,368.207,173.194,44.549,158.767
C02532=1038.144,377.746,368.273,173.182,44.543,158.765
C02533=1038.130,377.351,368.337,173.171,44.537,158.762
C02534=1038.117,376.957,368.404,173.158,44.531,158.759
C02535=1038.109,376.711,368.444,173.151,44.527,158.758
C02536=1038.099,376.464,368.485,173.144,44.524,158.756
C02537=1038.091,376.218,368.525,173.137,44.519,158.755
C02538=1038.083,375.972,368.566,173.130,44.516,158.753
C02539=1038.075,375.725,368.607,173.123,44.512,158.751
C02540=1038.066,375.478,368.648,173.115,44.508,158.750
C02541=1038.057,375.232,368.688,173.108,44.504,158.748
C02542=1038.049,374.985,368.729,173.101,44.501,158.747
C02543=1038.041,374.739,368.769,173.094,44.497,158.745
C02544=1038.032,374.492,368.810,173.087,44.494,158.743
C02545=1038.024,374.246,368.851,173.080,44.490,158.742
C02546=1038.015,373.999,368.891,173.073,44.486,158.740
C02547=1038.007,373.753,368.932,173.066,44.482,158.739
C02548=1037.999,373.507,368.973,173.059,44.478,158.737
C02549=1037.991,373.260,369.013,173.052,44.475,158.735
C02550=1037.983,373.013,369.054,173.046,44.471,158.734
C02551=1037.974,372.767,369.094,173.039,44.467,158.732
C02552=1037.966,372.520,369.134,173.032,44.464,158.731
C02553=1037.958,372.274,369.175,173.025,44.460,158.729
C02554=1037.950,372.027,369.215,173.018,44.456,158.728
C02555=1037.941,371.780,369.256,173.011,44.453,158.726
C02556=1037.933,371.534,369.295,173.004,44.449,158.725
C02557=1037.925,371.287,369.336,172.997,44.446,158.723
C02558=1037.917,371.041,369.376,172.991,44.442,158.722
C02559=1037.909,370.794,369.416,172.984,44.439,158.720
C02560=1037.900,370.547,369.457,172.977,44.435,158.719
C02561=1037.892,370.301,369.497,172.970,44.431,158.717
C02562=1037.884,370.054,369.537,172.963,44.428,158.716
C02563=1037.876,369.808,369.577,172.956,44.425,158.714
C02564=1037.868,369.561,369.616,172.950,44.421,158.713
C02565=1037.859,369.315,369.657,172.943,44.418,158.711
C02566=1037.851,369.068,369.696,172.936,44.414,158.710
C02567=1037.843,368.821,369.736,172.929,44.411,158.708
C02568=1037.835,368.574,369.776,172.922,44.407,158.707
C02569=1037.826,368.327,369.815,172.917,44.404,158.705
C02570=1037.817,368.081,369.855,172.909,44.400,158.704
C02571=1037.810,367.834,369.895,172.903,44.397,158.702
C02572=1037.801,367.588,369.935,172.896,44.394,158.701
C02573=1037.794,367.341,369.975,172.890,44.390,158.699
C02574=1037.785,367.094,370.014,172.883,44.387,158.698
C02575=1037.777,366.847,370.054,172.876,44.384,158.697
C02576=1037.769,366.601,370.093,172.869,44.381,158.695
C02577=1037.761,366.354,370.133,172.864,44.377,158.694
C02578=1037.753,366.107,370.172,172.857,44.374,158.692
C02579=1037.744,365.861,370.212,172.850,44.371,158.691
C02580=1037.737,365.614,370.251,172.843,44.368,158.690
C02581=1037.729,365.368,370.291,172.837,44.364,158.688
C02582=1037.721,365.121,370.330,172.830,44.361,158.687
C02583=1037.713,364.874,370.370,172.824,44.358,158.685
C02584=1037.705,364.627,370.409,172.818,44.354,158.684
C02585=1037.697,364.380,370.448,172.811,44.351,158.683
C02586=1037.688,364.134,370.488,172.805,44.348,158.681
C02587=1037.681,363.876,370.529,172.798,44.344,158.680
C02588=1037.672,363.619,370.570,172.791,44.341,158.678
C02589=1037.664,363.362,370.611,172.784,44.337,158.677
C02590=1037.655,363.105,370.652,172.778,44.334,158.675
C02591=1037.649,362.871,370.689,172.772,44.331,158.674
C02592=1037.641,362.637,370.726,172.766,44.328,158.673
C02593=1037.633,362.390,370.765,172.760,44.325,158.671
C02594=1037.625,362.143,370.804,172.753,44.322,158.670
C02595=1037.617,361.897,370.843,172.747,44.319,158.669
C02596=1037.609,361.649,370.883,172.740,44.316,158.667
C02597=1037.601,361.403,370.922,172.735,44.312,158.666
C02598=1037.593,361.156,370.960,172.728,44.309,158.665
C02599=1037.585,360.909,370.999,172.721,44.306,158.663
C02600=1037.577,360.663,371.038,172.716,44.303,158.662
C02601=1037.569,360.415,371.077,172.709,44.300,158.661
C02602=1037.562,360.169,371.115,172.703,44.297,158.659
C02603=1037.553,359.922,371.155,172.696,44.294,158.658
C02604=1037.545,359.675,371.193,172.691,44.291,158.657
C02605=1037.538,359.428,371.232,172.684,44.288,158.656
C02606=1037.530,359.181,371.270,172.678,44.285,158.654
C02607=1037.521,358.934,371.309,172.672,44.282,158.653
C02608=1037.514,358.688,371.348,172.666,44.279,158.652
C02609=1037.505,358.441,371.386,172.660,44.276,158.650
C02610=1037.498,358.194,371.425,172.654,44.273,158.649
C02611=1037.490,357.947,371.463,172.647,44.271,158.648
C02612=1037.483,357.700,371.502,172.642,44.267,158.647
C02613=1037.475,357.453,371.541,172.635,44.264,158.645
C02614=1037.467,357.206,371.579,172.629,44.261,158.644
C02615=1037.459,356.959,371.618,172.623,44.258,158.643
C02616=1037.451,356.712,371.656,172.617,44.256,158.642
C02617=1037.443,356.465,371.694,172.612,44.253,158.640
C02618=1037.435,356.218,371.733,172.605,44.250,158.639
C02619=1037.428,355.972,371.771,172.599,44.247,158.638
C02620=1037.420,355.724,371.810,172.593,44.244,158.636
C02621=1037.412,355.477,371.847,172.587,44.241,158.635
C02622=1037.405,355.231,371.886,172.581,44.239,158.634
C02623=1037.397,354.984,371.924,172.575,44.236,158.633
C02624=1037.388,354.737,371.962,172.569,44.232,158.632
C02625=1037.380,354.490,372.000,172.563,44.230,158.630
C02626=1037.373,354.243,372.038,172.557,44.227,158.629
C02627=1037.365,353.996,372.077,172.551,44.225,158.628
C02628=1037.358,353.749,372.114,172.545,44.221,158.627
C02629=1037.350,353.502,372.152,172.540,44.219,158.626
C02630=1037.342,353.255,372.191,172.533,44.216,158.624
C02631=1037.335,353.008,372.229,172.528,44.213,158.623
C02632=1037.326,352.761,372.267,172.522,44.211,158.622
C02633=1037.318,352.514,372.304,172.516,44.208,158.621
C02634=1037.311,352.267,372.342,172.510,44.205,158.620
C02635=1037.304,352.020,372.380,172.505,44.202,158.619
C02636=1037.295,351.773,372.419,172.498,44.200,158.617
C02637=1037.288,351.526,372.456,172.493,44.197,158.616
C02638=1037.281,351.279,372.494,172.487,44.194,158.615
C02639=1037.272,351.032,372.532,172.481,44.191,158.614
C02640=1037.265,350.785,372.569,172.475,44.189,158.612
C02641=1037.257,350.538,372.607,172.470,44.186,158.612
C02642=1037.250,350.291,372.645,172.464,44.184,158.610
C02643=1037.242,350.043,372.683,172.458,44.181,158.609
C02644=1037.234,349.797,372.720,172.452,44.178,158.608
C02645=1037.224,349.428,372.776,172.444,44.174,158.606
C02646=1037.212,349.061,372.832,172.435,44.170,158.604
C02647=1037.201,348.692,372.888,172.427,44.167,158.603
C02648=1037.189,348.324,372.944,172.419,44.163,158.601
C02649=1037.181,348.078,372.981,172.412,44.160,158.600
C02650=1037.174,347.830,373.019,172.407,44.158,158.599
C02651=1037.165,347.583,373.056,172.402,44.155,158.598
C02652=1037.158,347.336,373.094,172.396,44.152,158.597
C02653=1037.151,347.089,373.131,172.390,44.150,158.596
C02654=1037.143,346.842,373.168,172.384,44.148,158.595
C02655=1037.136,346.595,373.206,172.379,44.145,158.593
C02656=1037.128,346.348,373.243,172.374,44.143,158.592
C02657=1037.120,346.101,373.280,172.368,44.140,158.591
C02658=1037.113,345.854,373.318,172.363,44.138,158.590
C02659=1037.105,345.606,373.354,172.356,44.135,158.589
C02660=1037.098,345.359,373.391,172.351,44.132,158.588
C02661=1037.090,345.112,373.428,172.346,44.130,158.587
C02662=1037.083,344.865,373.466,172.340,44.127,158.586
C02663=1037.075,344.618,373.503,172.335,44.125,158.585
C02664=1037.068,344.371,373.540,172.330,44.122,158.584
C02665=1037.060,344.124,373.576,172.323,44.120,158.583
C02666=1037.053,343.877,373.614,172.318,44.118,158.581
C02667=1037.045,343.630,373.651,172.313,44.115,158.580
C02668=1037.038,343.382,373.688,172.307,44.113,158.579
C02669=1037.030,343.135,373.725,172.302,44.110,158.578
C02670=1037.023,342.887,373.761,172.297,44.108,158.577
C02671=1037.015,342.641,373.798,172.291,44.105,158.576
C02672=1037.008,342.393,373.836,172.286,44.103,158.575
C02673=1037.000,342.146,373.872,172.280,44.101,158.574
C02674=1036.993,341.899,373.910,172.274,44.099,158.573
C02675=1036.985,341.651,373.946,172.269,44.096,158.572
C02676=1036.978,341.404,373.983,172.264,44.094,158.571
C02677=1036.971,341.158,374.019,172.259,44.092,158.570
C02678=1036.963,340.911,374.056,172.253,44.089,158.569
C02679=1036.956,340.663,374.093,172.248,44.087,158.568
C02680=1036.948,340.416,374.129,172.243,44.085,158.567
C02681=1036.940,340.169,374.166,172.237,44.083,158.566
C02682=1036.933,339.921,374.202,172.232,44.080,158.565
C02683=1036.926,339.673,374.239,172.227,44.078,158.564
C02684=1036.919,339.427,374.275,172.222,44.076,158.563
C02685=1036.911,339.180,374.312,172.216,44.074,158.562
C02686=1036.903,338.932,374.348,172.211,44.071,158.561
C02687=1036.896,338.685,374.385,172.206,44.069,158.560
C02688=1036.888,338.437,374.421,172.201,44.067,158.559
C02689=1036.881,338.191,374.458,172.195,44.064,158.558
C02690=1036.873,337.944,374.494,172.190,44.062,158.557
C02691=1036.866,337.696,374.530,172.185,44.060,158.556
C02692=1036.859,337.448,374.567,172.180,44.058,158.555
C02693=1036.852,337.202,374.603,172.174,44.056,158.554
C02694=1036.844,336.954,374.639,172.169,44.053,158.553
C02695=1036.836,336.707,374.675,172.164,44.051,158.552
C02696=1036.829,336.459,374.712,172.159,44.049,158.551
C02697=1036.822,336.212,374.748,172.154,44.047,158.550
C02698=1036.815,335.965,374.784,172.149,44.045,158.549
C02699=1036.807,335.718,374.820,172.143,44.043,158.548
C02700=1036.800,335.471,374.856,172.138,44.041,158.547
C02701=1036.789,335.099,374.911,172.130,44.037,158.546
C02702=1036.778,334.727,374.965,172.122,44.034,158.544
C02703=1036.767,334.356,375.019,172.115,44.031,158.543
C02704=1036.756,333.984,375.073,172.107,44.028,158.542
C02705=1036.749,333.737,375.109,172.102,44.026,158.541
C02706=1036.741,333.490,375.145,172.097,44.024,158.540
C02707=1036.734,333.242,375.181,172.092,44.022,158.539
C02708=1036.727,332.995,375.217,172.086,44.020,158.538
C02709=1036.719,332.748,375.253,172.081,44.018,158.537
C02710=1036.712,332.500,375.288,172.076,44.016,158.536
C02711=1036.705,332.253,375.324,172.072,44.014,158.535
C02712=1036.697,332.006,375.360,172.067,44.012,158.534
C02713=1036.689,331.758,375.395,172.062,44.010,158.533
C02714=1036.682,331.511,375.431,172.057,44.008,158.532
C02715=1036.675,331.264,375.466,172.052,44.006,158.532
C02716=1036.667,331.016,375.503,172.046,44.004,158.531
C02717=1036.660,330.769,375.538,172.041,44.002,158.530
C02718=1036.653,330.522,375.574,172.036,44.000,158.529
C02719=1036.646,330.275,375.610,172.032,43.998,158.528
C02720=1036.639,330.027,375.645,172.027,43.996,158.527
C02721=1036.632,329.779,375.680,172.022,43.994,158.526
C02722=1036.624,329.532,375.716,172.017,43.992,158.525
C02723=1036.617,329.284,375.752,172.012,43.990,158.524
C02724=1036.610,329.038,375.788,172.007,43.988,158.523
C02725=1036.603,328.790,375.823,172.002,43.986,158.523
C02726=1036.596,328.543,375.859,171.997,43.984,158.522
C02727=1036.588,328.296,375.894,171.992,43.983,158.521
C02728=1036.581,328.048,375.929,171.987,43.980,158.520
C02729=1036.573,327.801,375.964,171.982,43.979,158.519
C02730=1036.566,327.553,375.999,171.977,43.977,158.518
C02731=1036.559,327.306,376.035,171.973,43.975,158.518
C02732=1036.551,327.058,376.070,171.968,43.973,158.517
C02733=1036.544,326.811,376.105,171.963,43.971,158.516
C02734=1036.536,326.564,376.140,171.958,43.970,158.515
C02735=1036.529,326.316,376.175,171.953,43.968,158.514
C02736=1036.522,326.069,376.210,171.948,43.966,158.513
C02737=1036.515,325.821,376.245,171.944,43.964,158.512
C02738=1036.507,325.573,376.280,171.939,43.963,158.512
C02739=1036.500,325.326,376.315,171.934,43.961,158.511
C02740=1036.492,325.079,376.349,171.929,43.959,158.510
C02741=1036.485,324.831,376.385,171.924,43.958,158.509
C02742=1036.477,324.584,376.419,171.920,43.955,158.508
C02743=1036.471,324.336,376.454,171.915,43.954,158.507
C02744=1036.463,324.089,376.489,171.910,43.952,158.507
C02745=1036.456,323.841,376.525,171.905,43.950,158.506
C02746=1036.448,323.594,376.559,171.901,43.949,158.505
C02747=1036.442,323.347,376.594,171.896,43.947,158.504
C02748=1036.433,323.099,376.629,171.891,43.945,158.503
C02749=1036.427,322.851,376.664,171.886,43.944,158.503
C02750=1036.419,322.604,376.698,171.882,43.942,158.502
C02751=1036.413,322.357,376.733,171.877,43.940,158.501
C02752=1036.405,322.109,376.768,171.872,43.939,158.500
C02753=1036.398,321.862,376.803,171.867,43.937,158.499
C02754=1036.391,321.614,376.837,171.863,43.935,158.499
C02755=1036.384,321.367,376.872,171.858,43.933,158.498
C02756=1036.376,321.120,376.907,171.853,43.932,158.497
C02757=1036.365,320.743,376.960,171.847,43.929,158.496
C02758=1036.355,320.367,377.012,171.839,43.927,158.495
C02759=1036.343,319.991,377.065,171.832,43.924,158.493
C02760=1036.333,319.615,377.117,171.825,43.922,158.492
C02761=1036.326,319.367,377.152,171.820,43.920,158.491
C02762=1036.318,319.119,377.187,171.816,43.918,158.491
C02763=1036.311,318.872,377.222,171.811,43.916,158.490
C02764=1036.304,318.624,377.255,171.806,43.915,158.489
C02765=1036.298,318.377,377.291,171.802,43.913,158.488
C02766=1036.290,318.129,377.324,171.797,43.911,158.487
C02767=1036.284,317.882,377.360,171.793,43.910,158.487
C02768=1036.276,317.634,377.393,171.789,43.909,158.486
C02769=1036.270,317.387,377.429,171.784,43.907,158.485
C02770=1036.262,317.139,377.462,171.779,43.905,158.484
C02771=1036.256,316.892,377.498,171.775,43.903,158.484
C02772=1036.248,316.644,377.531,171.770,43.902,158.483
C02773=1036.241,316.397,377.565,171.766,43.900,158.482
C02774=1036.234,316.149,377.600,171.761,43.899,158.481
C02775=1036.227,315.902,377.634,171.756,43.897,158.481
C02776=1036.221,315.655,377.669,171.752,43.895,158.480
C02777=1036.214,315.407,377.703,171.748,43.894,158.479
C02778=1036.207,315.159,377.737,171.744,43.892,158.478
C02779=1036.200,314.912,377.772,171.739,43.891,158.478
C02780=1036.193,314.665,377.805,171.735,43.889,158.477
C02781=1036.186,314.417,377.840,171.730,43.888,158.476
C02782=1036.179,314.169,377.874,171.725,43.886,158.475
C02783=1036.172,313.922,377.909,171.721,43.884,158.475
C02784=1036.166,313.675,377.942,171.716,43.883,158.474
C02785=1036.158,313.427,377.976,171.712,43.882,158.473
C02786=1036.152,313.179,378.011,171.707,43.880,158.472
C02787=1036.145,312.932,378.045,171.703,43.878,158.472
C02788=1036.138,312.684,378.080,171.699,43.877,158.471
C02789=1036.131,312.437,378.113,171.695,43.875,158.470
C02790=1036.125,312.189,378.147,171.690,43.874,158.470
C02791=1036.117,311.942,378.182,171.686,43.872,158.469
C02792=1036.110,311.694,378.216,171.681,43.871,158.468
C02793=1036.103,311.446,378.250,171.677,43.869,158.467
C02794=1036.096,311.198,378.283,171.673,43.868,158.467
C02795=1036.090,310.951,378.316,171.668,43.867,158.466
C02796=1036.082,310.704,378.350,171.664,43.865,158.465
C02797=1036.074,310.456,378.383,171.659,43.864,158.464
C02798=1036.067,310.209,378.417,171.655,43.863,158.464
C02799=1036.060,309.961,378.451,171.650,43.861,158.463
C02800=1036.053,309.714,378.484,171.646,43.860,158.462
C02801=1036.047,309.466,378.517,171.642,43.859,158.462
C02802=1036.039,309.218,378.551,171.638,43.857,158.461
C02803=1036.031,308.971,378.584,171.633,43.856,158.460
C02804=1036.024,308.723,378.618,171.628,43.855,158.460
C02805=1036.018,308.475,378.651,171.625,43.853,158.459
C02806=1036.011,308.228,378.685,171.620,43.852,158.459
C02807=1036.004,307.980,378.719,171.616,43.850,158.458
C02808=1035.996,307.733,378.752,171.611,43.849,158.457
C02809=1035.989,307.485,378.785,171.607,43.848,158.457
C02810=1035.982,307.237,378.819,171.603,43.847,158.456
C02811=1035.975,306.990,378.852,171.599,43.845,158.455
C02812=1035.969,306.742,378.885,171.594,43.844,158.454
C02813=1035.958,306.371,378.935,171.588,43.842,158.453
C02814=1035.947,305.999,378.985,171.582,43.840,158.452
C02815=1035.936,305.628,379.035,171.576,43.839,158.452
C02816=1035.926,305.257,379.085,171.569,43.837,158.451
C02817=1035.919,305.008,379.118,171.565,43.835,158.450
C02818=1035.912,304.761,379.151,171.561,43.834,158.449
C02819=1035.905,304.513,379.184,171.556,43.833,158.449
C02820=1035.897,304.266,379.218,171.552,43.831,158.448
C02821=1035.891,304.018,379.250,171.548,43.830,158.447
C02822=1035.884,303.771,379.284,171.544,43.829,158.447
C02823=1035.878,303.523,379.317,171.540,43.828,158.446
C02824=1035.870,303.276,379.350,171.535,43.827,158.445
C02825=1035.863,303.027,379.383,171.532,43.825,158.445
C02826=1035.856,302.780,379.416,171.527,43.824,158.444
C02827=1035.849,302.532,379.450,171.523,43.823,158.443
C02828=1035.843,302.284,379.483,171.519,43.821,158.443
C02829=1035.835,302.037,379.516,171.514,43.820,158.442
C02830=1035.829,301.790,379.549,171.511,43.819,158.442
C02831=1035.822,301.541,379.582,171.506,43.818,158.441
C02832=1035.815,301.294,379.615,171.502,43.817,158.440
C02833=1035.808,301.046,379.648,171.499,43.815,158.440
C02834=1035.801,300.799,379.680,171.494,43.814,158.439
C02835=1035.794,300.550,379.713,171.490,43.813,158.438
C02836=1035.788,300.303,379.747,171.485,43.812,158.438
C02837=1035.780,300.055,379.779,171.482,43.811,158.437
C02838=1035.774,299.808,379.812,171.478,43.809,158.437
C02839=1035.768,299.560,379.845,171.473,43.808,158.436
C02840=1035.761,299.312,379.878,171.469,43.807,158.435
C02841=1035.753,299.065,379.911,171.466,43.806,158.435
C02842=1035.747,298.817,379.944,171.461,43.805,158.434
C02843=1035.740,298.569,379.977,171.457,43.804,158.434
C02844=1035.734,298.322,380.009,171.454,43.802,158.433
C02845=1035.726,298.074,380.042,171.449,43.801,158.432
C02846=1035.720,297.826,380.075,171.445,43.800,158.432
C02847=1035.713,297.578,380.108,171.441,43.799,158.431
C02848=1035.707,297.330,380.141,171.438,43.797,158.430
C02849=1035.700,297.083,380.173,171.433,43.796,158.430
C02850=1035.693,296.835,380.207,171.429,43.795,158.429
C02851=1035.686,296.588,380.239,171.426,43.794,158.429
C02852=1035.680,296.340,380.272,171.421,43.793,158.428
C02853=1035.672,296.092,380.305,171.417,43.792,158.427
C02854=1035.666,295.845,380.337,171.414,43.791,158.427
C02855=1035.660,295.597,380.370,171.410,43.790,158.426
C02856=1035.653,295.349,380.401,171.405,43.789,158.426
C02857=1035.646,295.101,380.435,171.401,43.787,158.425
C02858=1035.640,294.853,380.467,171.398,43.786,158.425
C02859=1035.633,294.606,380.499,171.393,43.785,158.424
C02860=1035.626,294.358,380.533,171.389,43.784,158.423
C02861=1035.619,294.110,380.565,171.386,43.783,158.423
C02862=1035.612,293.862,380.596,171.382,43.782,158.422
C02863=1035.605,293.614,380.629,171.377,43.781,158.422
C02864=1035.598,293.367,380.661,171.374,43.780,158.421
C02865=1035.592,293.119,380.694,171.370,43.779,158.421
C02866=1035.585,292.871,380.726,171.365,43.778,158.420
C02867=1035.578,292.623,380.758,171.362,43.777,158.419
C02868=1035.571,292.376,380.791,171.358,43.776,158.419
C02869=1035.562,292.021,380.836,171.352,43.774,158.418
C02870=1035.552,291.667,380.883,171.347,43.773,158.417
C02871=1035.541,291.311,380.929,171.341,43.772,158.417
C02872=1035.532,290.957,380.974,171.336,43.770,158.416
C02873=1035.525,290.709,381.007,171.332,43.769,158.415
C02874=1035.518,290.462,381.038,171.328,43.768,158.415
C02875=1035.512,290.214,381.071,171.325,43.767,158.414
C02876=1035.505,289.966,381.102,171.320,43.767,158.414
C02877=1035.497,289.718,381.135,171.316,43.765,158.413
C02878=1035.491,289.470,381.166,171.313,43.764,158.412
C02879=1035.484,289.223,381.199,171.309,43.763,158.412
C02880=1035.478,288.975,381.230,171.304,43.762,158.411
C02881=1035.471,288.727,381.262,171.301,43.762,158.411
C02882=1035.463,288.479,381.294,171.297,43.760,158.410
C02883=1035.456,288.232,381.326,171.294,43.760,158.410
C02884=1035.450,287.983,381.358,171.290,43.759,158.409
C02885=1035.444,287.735,381.390,171.286,43.758,158.409
C02886=1035.437,287.488,381.422,171.282,43.757,158.408
C02887=1035.430,287.240,381.453,171.278,43.756,158.408
C02888=1035.422,286.992,381.485,171.275,43.755,158.407
C02889=1035.415,286.744,381.517,171.271,43.754,158.407
C02890=1035.409,286.496,381.549,171.266,43.753,158.406
C02891=1035.403,286.248,381.581,171.263,43.752,158.406
C02892=1035.396,286.000,381.612,171.259,43.752,158.405
C02893=1035.389,285.752,381.644,171.256,43.751,158.404
C02894=1035.382,285.505,381.676,171.252,43.750,158.404
C02895=1035.376,285.257,381.707,171.249,43.749,158.404
C02896=1035.367,285.009,381.738,171.244,43.748,158.403
C02897=1035.361,284.761,381.770,171.240,43.747,158.403
C02898=1035.354,284.513,381.801,171.237,43.747,158.402
C02899=1035.347,284.265,381.833,171.233,43.746,158.401
C02900=1035.341,284.017,381.864,171.230,43.745,158.401
C02901=1035.334,283.769,381.896,171.225,43.744,158.401
C02902=1035.327,283.522,381.928,171.222,43.743,158.400
C02903=1035.320,283.274,381.959,171.218,43.742,158.400
C02904=1035.313,283.026,381.991,171.215,43.742,158.399
C02905=1035.307,282.778,382.022,171.211,43.741,158.398
C02906=1035.300,282.531,382.053,171.207,43.740,158.398
C02907=1035.293,282.283,382.085,171.204,43.739,158.398
C02908=1035.286,282.035,382.116,171.199,43.738,158.397
C02909=1035.280,281.787,382.148,171.196,43.737,158.397
C02910=1035.273,281.539,382.179,171.192,43.737,158.396
C02911=1035.266,281.291,382.211,171.189,43.736,158.396
C02912=1035.260,281.043,382.242,171.185,43.735,158.395
C02913=1035.253,280.795,382.273,171.182,43.734,158.395
C02914=1035.246,280.547,382.304,171.178,43.734,158.394
C02915=1035.240,280.299,382.336,171.175,43.733,158.394
C02916=1035.233,280.051,382.367,171.171,43.732,158.393
C02917=1035.226,279.803,382.399,171.167,43.731,158.393
C02918=1035.219,279.555,382.430,171.163,43.730,158.392
C02919=1035.213,279.307,382.461,171.159,43.730,158.392
C02920=1035.205,279.060,382.492,171.156,43.729,158.391
C02921=1035.199,278.811,382.523,171.152,43.728,158.391
C02922=1035.192,278.563,382.554,171.149,43.727,158.390
C02923=1035.185,278.315,382.586,171.145,43.727,158.390
C02924=1035.179,278.067,382.617,171.142,43.726,158.389
C02925=1035.170,277.724,382.660,171.137,43.725,158.389
C02926=1035.160,277.382,382.702,171.131,43.724,158.388
C02927=1035.151,277.040,382.745,171.127,43.723,158.387
C02928=1035.142,276.697,382.788,171.122,43.722,158.387
C02929=1035.135,276.449,382.820,171.118,43.721,158.386
C02930=1035.128,276.201,382.850,171.115,43.720,158.386
C02931=1035.121,275.953,382.881,171.111,43.720,158.385
C02932=1035.115,275.705,382.912,171.108,43.719,158.385
C02933=1035.107,275.457,382.943,171.104,43.718,158.385
C02934=1035.101,275.209,382.974,171.101,43.717,158.384
C02935=1035.095,274.961,383.005,171.097,43.716,158.384
C02936=1035.087,274.714,383.035,171.094,43.716,158.383
C02937=1035.081,274.465,383.066,171.090,43.715,158.383
C02938=1035.074,274.217,383.098,171.086,43.715,158.382
C02939=1035.067,273.969,383.128,171.082,43.714,158.382
C02940=1035.060,273.721,383.159,171.079,43.713,158.381
C02941=1035.054,273.473,383.190,171.075,43.713,158.381
C02942=1035.047,273.225,383.220,171.072,43.712,158.380
C02943=1035.041,272.977,383.251,171.068,43.711,158.380
C02944=1035.034,272.729,383.282,171.065,43.711,158.380
C02945=1035.027,272.481,383.313,171.061,43.710,158.379
C02946=1035.020,272.233,383.343,171.058,43.709,158.379
C02947=1035.013,271.986,383.374,171.054,43.709,158.378
C02948=1035.007,271.737,383.404,171.051,43.708,158.378
C02949=1035.001,271.489,383.435,171.047,43.707,158.377
C02950=1034.993,271.241,383.466,171.044,43.707,158.377
C02951=1034.987,270.993,383.496,171.040,43.706,158.376
C02952=1034.980,270.745,383.526,171.037,43.706,158.376
C02953=1034.974,270.497,383.557,171.034,43.705,158.376
C02954=1034.966,270.249,383.588,171.030,43.705,158.375
C02955=1034.960,270.001,383.618,171.027,43.704,158.375
C02956=1034.953,269.753,383.649,171.023,43.703,158.374
C02957=1034.946,269.505,383.679,171.020,43.703,158.374
C02958=1034.939,269.257,383.710,171.016,43.702,158.374
C02959=1034.933,269.009,383.740,171.013,43.701,158.373
C02960=1034.926,268.761,383.771,171.009,43.701,158.373
C02961=1034.919,268.513,383.801,171.006,43.701,158.372
C02962=1034.913,268.264,383.831,171.003,43.700,158.372
C02963=1034.906,268.017,383.861,171.000,43.699,158.372
C02964=1034.899,267.768,383.891,170.996,43.698,158.371
C02965=1034.892,267.520,383.923,170.993,43.698,158.371
C02966=1034.886,267.273,383.952,170.990,43.697,158.370
C02967=1034.879,267.024,383.983,170.986,43.697,158.370
C02968=1034.872,266.776,384.013,170.983,43.696,158.369
C02969=1034.866,266.529,384.043,170.979,43.696,158.369
C02970=1034.859,266.280,384.074,170.976,43.695,158.369
C02971=1034.852,266.032,384.104,170.973,43.695,158.368
C02972=1034.845,265.784,384.134,170.969,43.694,158.368
C02973=1034.839,265.536,384.164,170.966,43.694,158.367
C02974=1034.832,265.288,384.194,170.962,43.693,158.367
C02975=1034.825,265.040,384.224,170.959,43.693,158.367
C02976=1034.818,264.792,384.254,170.955,43.692,158.366
C02977=1034.812,264.543,384.284,170.952,43.691,158.366
C02978=1034.806,264.295,384.314,170.948,43.691,158.365
C02979=1034.798,264.047,384.344,170.945,43.691,158.365
C02980=1034.791,263.799,384.374,170.943,43.690,158.365
C02981=1034.783,263.461,384.416,170.938,43.689,158.364
C02982=1034.773,263.123,384.456,170.933,43.688,158.364
C02983=1034.764,262.785,384.497,170.929,43.688,158.363
C02984=1034.756,262.448,384.538,170.924,43.687,158.363
C02985=1034.749,262.199,384.568,170.921,43.687,158.362
C02986=1034.742,261.951,384.598,170.917,43.686,158.362
C02987=1034.735,261.704,384.628,170.914,43.685,158.361
C02988=1034.729,261.454,384.658,170.911,43.685,158.361
C02989=1034.723,261.207,384.688,170.907,43.685,158.361
C02990=1034.715,260.959,384.717,170.904,43.684,158.360
C02991=1034.708,260.710,384.747,170.900,43.684,158.360
C02992=1034.701,260.463,384.777,170.897,43.684,158.360
C02993=1034.694,260.214,384.806,170.895,43.683,158.359
C02994=1034.688,259.966,384.836,170.891,43.683,158.359
C02995=1034.681,259.718,384.866,170.888,43.682,158.358
C02996=1034.674,259.469,384.895,170.885,43.682,158.358
C02997=1034.667,259.222,384.925,170.881,43.681,158.358
C02998=1034.660,258.973,384.954,170.878,43.681,158.357
C02999=1034.653,258.726,384.984,170.875,43.681,158.357
C03000=1034.646,258.477,385.013,170.871,43.681,158.357
C03001=1034.640,258.229,385.043,170.868,43.680,158.356
C03002=1034.633,257.981,385.072,170.865,43.680,158.356
C03003=1034.626,257.732,385.102,170.862,43.679,158.356
C03004=1034.619,257.484,385.131,170.859,43.679,158.355
C03005=1034.612,257.236,385.161,170.855,43.678,158.355
C03006=1034.605,256.988,385.190,170.852,43.678,158.355
C03007=1034.598,256.740,385.220,170.849,43.678,158.354
C03008=1034.592,256.492,385.249,170.845,43.678,158.354
C03009=1034.585,256.243,385.278,170.842,43.677,158.353
C03010=1034.578,255.996,385.308,170.840,43.677,158.353
C03011=1034.572,255.747,385.338,170.836,43.676,158.353
C03012=1034.565,255.499,385.367,170.833,43.676,158.352
C03013=1034.557,255.251,385.396,170.830,43.676,158.352
C03014=1034.551,255.003,385.425,170.826,43.675,158.352
C03015=1034.545,254.755,385.455,170.823,43.675,158.351
C03016=1034.538,254.506,385.484,170.820,43.674,158.351
C03017=1034.532,254.258,385.513,170.817,43.674,158.351
C03018=1034.524,254.010,385.543,170.814,43.673,158.350
C03019=1034.518,253.762,385.573,170.810,43.673,158.350
C03020=1034.511,253.513,385.601,170.807,43.673,158.350
C03021=1034.504,253.266,385.631,170.804,43.673,158.349
C03022=1034.498,253.018,385.660,170.801,43.672,158.349
C03023=1034.491,252.769,385.690,170.798,43.672,158.349
C03024=1034.485,252.521,385.719,170.795,43.672,158.348
C03025=1034.478,252.272,385.749,170.791,43.671,158.348
C03026=1034.471,252.024,385.778,170.788,43.671,158.348
C03027=1034.464,251.776,385.806,170.785,43.670,158.347
C03028=1034.457,251.528,385.836,170.782,43.670,158.347
C03029=1034.451,251.279,385.865,170.779,43.670,158.347
C03030=1034.445,251.032,385.894,170.775,43.669,158.346
C03031=1034.438,250.783,385.924,170.773,43.669,158.346
C03032=1034.432,250.535,385.953,170.770,43.668,158.346
C03033=1034.425,250.287,385.981,170.766,43.668,158.345
C03034=1034.418,250.038,386.011,170.763,43.668,158.345
C03035=1034.411,249.790,386.040,170.761,43.667,158.345
C03036=1034.405,249.542,386.069,170.757,43.667,158.344
C03037=1034.396,249.203,386.109,170.753,43.667,158.344
C03038=1034.387,248.864,386.148,170.748,43.666,158.343
C03039=1034.378,248.524,386.188,170.745,43.666,158.343
C03040=1034.368,248.185,386.228,170.740,43.665,158.342
C03041=1034.362,247.937,386.258,170.737,43.665,158.342
C03042=1034.355,247.688,386.287,170.734,43.664,158.342
C03043=1034.349,247.440,386.316,170.731,43.664,158.341
C03044=1034.343,247.192,386.345,170.728,43.664,158.341
C03045=1034.336,246.943,386.374,170.725,43.663,158.341
C03046=1034.329,246.696,386.402,170.722,43.663,158.340
C03047=1034.323,246.447,386.432,170.719,43.663,158.340
C03048=1034.317,246.199,386.461,170.716,43.662,158.340
C03049=1034.310,245.950,386.490,170.712,43.662,158.339
C03050=1034.303,245.702,386.519,170.710,43.661,158.339
C03051=1034.296,245.454,386.547,170.707,43.661,158.339
C03052=1034.290,245.206,386.577,170.703,43.661,158.338
C03053=1034.284,244.958,386.606,170.701,43.661,158.338
C03054=1034.277,244.709,386.634,170.698,43.660,158.338
C03055=1034.270,244.461,386.663,170.694,43.660,158.338
C03056=1034.264,244.213,386.692,170.692,43.660,158.337
C03057=1034.257,243.965,386.720,170.689,43.659,158.337
C03058=1034.251,243.717,386.749,170.685,43.659,158.337
C03059=1034.244,243.467,386.778,170.682,43.659,158.336
C03060=1034.237,243.220,386.806,170.680,43.659,158.336
C03061=1034.231,242.971,386.835,170.676,43.658,158.336
C03062=1034.224,242.724,386.864,170.673,43.658,158.335
C03063=1034.217,242.475,386.893,170.671,43.658,158.335
C03064=1034.211,242.226,386.921,170.668,43.658,158.335
C03065=1034.204,241.978,386.950,170.664,43.657,158.334
C03066=1034.197,241.730,386.978,170.662,43.657,158.334
C03067=1034.191,241.482,387.007,170.659,43.657,158.334
C03068=1034.184,241.234,387.035,170.655,43.657,158.334
C03069=1034.178,240.985,387.065,170.653,43.657,158.333
C03070=1034.171,240.737,387.092,170.650,43.656,158.333
C03071=1034.165,240.488,387.121,170.646,43.656,158.333
C03072=1034.158,240.241,387.150,170.644,43.656,158.332
C03073=1034.152,239.992,387.178,170.641,43.656,158.332
C03074=1034.145,239.744,387.207,170.638,43.656,158.332
C03075=1034.138,239.496,387.234,170.635,43.655,158.331
C03076=1034.131,239.247,387.263,170.632,43.655,158.331
C03077=1034.125,238.998,387.291,170.629,43.655,158.331
C03078=1034.118,238.750,387.320,170.627,43.655,158.331
C03079=1034.111,238.502,387.348,170.623,43.654,158.330
C03080=1034.105,238.254,387.377,170.620,43.654,158.330
C03081=1034.098,238.005,387.404,170.618,43.654,158.330
C03082=1034.091,237.758,387.433,170.614,43.654,158.329
C03083=1034.084,237.509,387.461,170.611,43.654,158.329
C03084=1034.077,237.260,387.490,170.609,43.654,158.329
C03085=1034.071,237.012,387.518,170.606,43.654,158.329
C03086=1034.064,236.764,387.546,170.602,43.653,158.328
C03087=1034.057,236.516,387.574,170.600,43.653,158.328
C03088=1034.051,236.267,387.602,170.597,43.653,158.328
C03089=1034.044,236.019,387.631,170.594,43.653,158.328
C03090=1034.037,235.771,387.658,170.591,43.653,158.327
C03091=1034.031,235.522,387.686,170.588,43.653,158.327
C03092=1034.024,235.274,387.715,170.586,43.653,158.327
C03093=1034.015,234.929,387.754,170.581,43.652,158.326
C03094=1034.005,234.583,387.793,170.577,43.652,158.326
C03095=1033.997,234.238,387.832,170.574,43.651,158.325
C03096=1033.987,233.892,387.871,170.569,43.652,158.325
C03097=1033.980,233.645,387.899,170.566,43.652,158.325
C03098=1033.973,233.396,387.927,170.564,43.651,158.325
C03099=1033.967,233.147,387.955,170.561,43.651,158.324
C03100=1033.960,232.900,387.984,170.558,43.651,158.324
C03101=1033.954,232.651,388.012,170.555,43.651,158.324
C03102=1033.947,232.403,388.039,170.552,43.651,158.324
C03103=1033.940,232.154,388.067,170.550,43.651,158.323
C03104=1033.934,231.906,388.095,170.546,43.651,158.323
C03105=1033.927,231.658,388.124,170.544,43.650,158.323
C03106=1033.921,231.409,388.151,170.541,43.650,158.322
C03107=1033.914,231.161,388.179,170.539,43.650,158.322
C03108=1033.907,230.912,388.207,170.535,43.650,158.322
C03109=1033.901,230.664,388.235,170.532,43.650,158.322
C03110=1033.894,230.416,388.262,170.530,43.650,158.321
C03111=1033.887,230.167,388.290,170.526,43.649,158.321
C03112=1033.880,229.919,388.319,170.524,43.649,158.321
C03113=1033.874,229.671,388.346,170.521,43.649,158.321
C03114=1033.867,229.422,388.374,170.518,43.649,158.320
C03115=1033.860,229.174,388.402,170.515,43.649,158.320
C03116=1033.854,228.925,388.430,170.512,43.649,158.320
C03117=1033.848,228.677,388.458,170.510,43.649,158.320
C03118=1033.841,228.428,388.486,170.507,43.648,158.319
C03119=1033.835,228.181,388.513,170.504,43.648,158.319
C03120=1033.828,227.932,388.541,170.501,43.648,158.319
C03121=1033.821,227.684,388.568,170.499,43.648,158.319
C03122=1033.814,227.436,388.596,170.496,43.648,158.318
C03123=1033.807,227.187,388.623,170.493,43.648,158.318
C03124=1033.801,226.939,388.651,170.490,43.648,158.318
C03125=1033.794,226.690,388.679,170.487,43.648,158.318
C03126=1033.787,226.442,388.706,170.485,43.648,158.317
C03127=1033.780,226.193,388.733,170.482,43.648,158.317
C03128=1033.774,225.945,388.761,170.479,43.648,158.317
C03129=1033.767,225.696,388.788,170.476,43.648,158.317
C03130=1033.760,225.448,388.816,170.474,43.648,158.316
C03131=1033.753,225.199,388.844,170.471,43.648,158.316
C03132=1033.746,224.951,388.871,170.468,43.648,158.316
C03133=1033.739,224.703,388.899,170.465,43.647,158.316
C03134=1033.734,224.454,388.925,170.462,43.647,158.315
C03135=1033.727,224.206,388.953,170.460,43.648,158.315
C03136=1033.720,223.957,388.981,170.457,43.648,158.315
C03137=1033.714,223.709,389.008,170.455,43.647,158.315
C03138=1033.706,223.461,389.036,170.451,43.647,158.314
C03139=1033.700,223.212,389.063,170.449,43.647,158.314
C03140=1033.693,222.963,389.090,170.446,43.647,158.314
C03141=1033.687,222.716,389.118,170.444,43.647,158.314
C03142=1033.680,222.467,389.145,170.440,43.647,158.314
C03143=1033.673,222.218,389.172,170.438,43.647,158.313
C03144=1033.667,221.970,389.200,170.435,43.647,158.313
C03145=1033.660,221.722,389.227,170.433,43.647,158.313
C03146=1033.653,221.473,389.254,170.429,43.647,158.312
C03147=1033.647,221.225,389.281,170.427,43.647,158.312
C03148=1033.640,220.977,389.309,170.424,43.647,158.312
C03149=1033.631,220.624,389.348,170.421,43.647,158.312
C03150=1033.621,220.271,389.386,170.416,43.646,158.311
C03151=1033.612,219.918,389.426,170.413,43.646,158.311
C03152=1033.602,219.565,389.464,170.409,43.646,158.311
C03153=1033.596,219.316,389.491,170.407,43.646,158.310
C03154=1033.588,219.068,389.518,170.404,43.647,158.310
C03155=1033.582,218.820,389.545,170.401,43.647,158.310
C03156=1033.575,218.572,389.572,170.398,43.646,158.310
C03157=1033.569,218.323,389.600,170.396,43.647,158.310
C03158=1033.561,218.074,389.626,170.393,43.647,158.309
C03159=1033.555,217.826,389.654,170.391,43.647,158.309
C03160=1033.548,217.578,389.680,170.387,43.646,158.309
C03161=1033.542,217.330,389.708,170.385,43.647,158.309
C03162=1033.534,217.081,389.734,170.382,43.647,158.309
C03163=1033.528,216.832,389.761,170.380,43.646,158.308
C03164=1033.522,216.584,389.788,170.377,43.647,158.308
C03165=1033.515,216.335,389.815,170.374,43.647,158.308
C03166=1033.508,216.087,389.843,170.372,43.647,158.308
C03167=1033.501,215.838,389.869,170.369,43.647,158.308
C03168=1033.495,215.590,389.896,170.367,43.647,158.307
C03169=1033.488,215.342,389.923,170.364,43.647,158.307
C03170=1033.482,215.092,389.950,170.362,43.647,158.307
C03171=1033.474,214.844,389.977,170.358,43.647,158.307
C03172=1033.468,214.596,390.004,170.356,43.647,158.306
C03173=1033.461,214.348,390.031,170.353,43.647,158.306
C03174=1033.455,214.099,390.058,170.351,43.647,158.306
C03175=1033.448,213.851,390.084,170.349,43.647,158.306
C03176=1033.441,213.602,390.111,170.345,43.647,158.305
C03177=1033.434,213.354,390.138,170.343,43.647,158.305
C03178=1033.428,213.104,390.165,170.340,43.647,158.305
C03179=1033.421,212.857,390.192,170.338,43.647,158.305
C03180=1033.415,212.608,390.219,170.336,43.647,158.305
C03181=1033.408,212.359,390.245,170.333,43.647,158.304
C03182=1033.401,212.112,390.272,170.330,43.647,158.304
C03183=1033.394,211.863,390.299,170.327,43.647,158.304
C03184=1033.389,211.614,390.326,170.325,43.647,158.304
C03185=1033.381,211.366,390.352,170.323,43.647,158.304
C03186=1033.374,211.118,390.379,170.319,43.647,158.303
C03187=1033.368,210.869,390.406,170.317,43.647,158.303
C03188=1033.361,210.620,390.432,170.314,43.647,158.303
C03189=1033.354,210.372,390.459,170.312,43.648,158.303
C03190=1033.348,210.123,390.485,170.310,43.647,158.303
C03191=1033.341,209.875,390.512,170.307,43.647,158.302
C03192=1033.334,209.626,390.539,170.305,43.648,158.302
C03193=1033.328,209.378,390.565,170.301,43.648,158.302
C03194=1033.321,209.129,390.592,170.299,43.648,158.302
C03195=1033.314,208.881,390.618,170.297,43.648,158.302
C03196=1033.308,208.632,390.645,170.294,43.648,158.301
C03197=1033.301,208.383,390.671,170.292,43.648,158.301
C03198=1033.294,208.135,390.697,170.289,43.648,158.301
C03199=1033.287,207.887,390.724,170.287,43.648,158.301
C03200=1033.281,207.638,390.752,170.284,43.648,158.301
C03201=1033.274,207.390,390.778,170.281,43.648,158.300
C03202=1033.267,207.141,390.804,170.279,43.648,158.300
C03203=1033.260,206.893,390.830,170.276,43.648,158.300
C03204=1033.253,206.645,390.856,170.274,43.649,158.300
C03205=1033.244,206.297,390.893,170.270,43.649,158.300
C03206=1033.235,205.951,390.930,170.266,43.649,158.299
C03207=1033.225,205.603,390.967,170.263,43.649,158.299
C03208=1033.216,205.256,391.003,170.260,43.649,158.299
C03209=1033.190,204.206,391.109,169.924,43.545,158.249
C03210=1033.184,203.958,391.134,169.921,43.546,158.249
C03211=1033.177,203.709,391.159,169.917,43.546,158.249
C03212=1033.172,203.461,391.184,169.914,43.547,158.249
C03213=1033.166,203.212,391.209,169.910,43.548,158.249
C03214=1033.160,202.963,391.234,169.907,43.549,158.249
C03215=1033.153,202.714,391.260,169.903,43.550,158.249
C03216=1033.147,202.465,391.284,169.900,43.551,158.249
C03217=1033.141,202.217,391.309,169.896,43.552,158.249
C03218=1033.135,201.969,391.334,169.893,43.552,158.248
C03219=1033.129,201.719,391.359,169.889,43.554,158.248
C03220=1033.123,201.471,391.384,169.886,43.554,158.248
C03221=1033.117,201.223,391.409,169.882,43.555,158.248
C03222=1033.111,200.974,391.434,169.879,43.556,158.248
C03223=1033.104,200.725,391.458,169.875,43.557,158.248
C03224=1033.099,200.476,391.483,169.872,43.557,158.248
C03225=1033.093,200.228,391.508,169.869,43.559,158.248
C03226=1033.086,199.979,391.532,169.866,43.560,158.248
C03227=1033.080,199.730,391.557,169.862,43.561,158.248
C03228=1033.074,199.481,391.581,169.859,43.562,158.248
C03229=1033.068,199.233,391.606,169.855,43.563,158.247
C03230=1033.061,198.984,391.630,169.852,43.564,158.247
C03231=1033.055,198.735,391.655,169.848,43.565,158.247
C03232=1033.048,198.487,391.680,169.845,43.566,158.247
C03233=1033.043,198.238,391.704,169.841,43.566,158.247
C03234=1033.036,197.989,391.728,169.838,43.568,158.247
C03235=1033.030,197.740,391.753,169.834,43.569,158.247
C03236=1033.024,197.492,391.777,169.831,43.570,158.247
C03237=1033.018,197.243,391.802,169.827,43.571,158.247
C03238=1033.012,196.994,391.827,169.824,43.572,158.247
C03239=1033.005,196.745,391.851,169.821,43.573,158.247
C03240=1033.000,196.497,391.875,169.818,43.574,158.247
C03241=1032.993,196.248,391.900,169.815,43.575,158.247
C03242=1032.987,195.999,391.925,169.811,43.576,158.247
C03243=1032.981,195.751,391.948,169.808,43.577,158.246
C03244=1032.975,195.501,391.973,169.804,43.578,158.246
C03245=1032.968,195.253,391.998,169.801,43.579,158.246
C03246=1032.963,195.005,392.022,169.797,43.580,158.246
C03247=1032.957,194.756,392.046,169.794,43.581,158.246
C03248=1032.951,194.506,392.071,169.790,43.582,158.246
C03249=1032.944,194.259,392.095,169.787,43.583,158.246
C03250=1032.938,194.009,392.120,169.785,43.584,158.246
C03251=1032.932,193.761,392.143,169.781,43.585,158.246
C03252=1032.926,193.512,392.167,169.778,43.586,158.246
C03253=1032.920,193.263,392.192,169.774,43.588,158.246
C03254=1032.914,193.015,392.215,169.771,43.588,158.246
C03255=1032.908,192.766,392.241,169.768,43.589,158.246
C03256=1032.902,192.518,392.264,169.764,43.591,158.246
C03257=1032.896,192.268,392.289,169.761,43.591,158.246
C03258=1032.890,192.020,392.313,169.757,43.593,158.246
C03259=1032.884,191.771,392.337,169.755,43.594,158.246
C03260=1032.877,191.522,392.361,169.752,43.594,158.245
C03261=1032.872,191.273,392.386,169.748,43.596,158.245
C03262=1032.865,191.024,392.410,169.745,43.597,158.245
C03263=1032.860,190.776,392.434,169.741,43.598,158.245
C03264=1032.853,190.527,392.458,169.738,43.599,158.245
C03265=1032.848,190.278,392.482,169.735,43.600,158.245
C03266=1032.841,190.029,392.506,169.731,43.601,158.245
C03267=1032.836,189.780,392.531,169.728,43.602,158.245
C03268=1032.829,189.531,392.555,169.725,43.603,158.245
C03269=1032.824,189.283,392.579,169.721,43.604,158.245
C03270=1032.817,189.000,392.606,169.719,43.605,158.245
C03271=1032.810,188.716,392.634,169.715,43.607,158.245
C03272=1032.803,188.431,392.661,169.711,43.608,158.245
C03273=1032.796,188.148,392.689,169.707,43.609,158.245
C03274=1032.791,187.899,392.713,169.704,43.610,158.245
C03275=1032.784,187.650,392.737,169.700,43.611,158.245
C03276=1032.779,187.402,392.761,169.697,43.613,158.245
C03277=1032.772,187.153,392.785,169.694,43.613,158.244
C03278=1032.766,186.904,392.809,169.692,43.614,158.244
C03279=1032.761,186.656,392.833,169.688,43.616,158.244
C03280=1032.754,186.406,392.856,169.685,43.616,158.244
C03281=1032.749,186.158,392.881,169.682,43.617,158.244
C03282=1032.742,185.909,392.905,169.678,43.619,158.244
C03283=1032.737,185.660,392.929,169.675,43.620,158.244
C03284=1032.731,185.412,392.953,169.672,43.621,158.244
C03285=1032.725,185.162,392.977,169.668,43.622,158.244
C03286=1032.719,184.914,393.001,169.665,43.623,158.244
C03287=1032.713,184.665,393.024,169.662,43.624,158.244
C03288=1032.708,184.416,393.049,169.660,43.625,158.244
C03289=1032.702,184.168,393.072,169.656,43.626,158.244
C03290=1032.696,183.919,393.096,169.653,43.628,158.244
C03291=1032.690,183.670,393.120,169.650,43.628,158.244
C03292=1032.685,183.421,393.144,169.647,43.629,158.244
C03293=1032.679,183.173,393.168,169.643,43.631,158.244
C03294=1032.672,182.924,393.192,169.640,43.632,158.244
C03295=1032.666,182.675,393.215,169.638,43.633,158.244
C03296=1032.660,182.426,393.239,169.634,43.634,158.244
C03297=1032.654,182.177,393.262,169.631,43.636,158.244
C03298=1032.646,181.928,393.285,169.628,43.637,158.244
C03299=1032.641,181.679,393.308,169.624,43.638,158.244
C03300=1032.635,181.431,393.332,169.621,43.639,158.244
C03301=1032.628,181.182,393.355,169.619,43.641,158.244
C03302=1032.622,180.933,393.379,169.615,43.642,158.244
C03303=1032.616,180.684,393.402,169.612,43.643,158.244
C03304=1032.610,180.435,393.426,169.609,43.644,158.244
C03305=1032.603,180.187,393.448,169.606,43.647,158.244
C03306=1032.597,179.938,393.472,169.603,43.648,158.244
C03307=1032.591,179.689,393.495,169.600,43.649,158.244
C03308=1032.585,179.440,393.518,169.596,43.650,158.244
C03309=1032.579,179.191,393.542,169.593,43.652,158.244
C03310=1032.573,178.942,393.565,169.590,43.653,158.244
C03311=1032.566,178.693,393.588,169.587,43.654,158.244
C03312=1032.560,178.445,393.611,169.584,43.655,158.244
C03313=1032.554,178.196,393.634,169.581,43.657,158.244
C03314=1032.548,177.947,393.658,169.578,43.658,158.244
C03315=1032.542,177.698,393.681,169.574,43.659,158.244
C03316=1032.536,177.449,393.704,169.571,43.660,158.244
C03317=1032.529,177.201,393.727,169.569,43.662,158.244
C03318=1032.523,176.951,393.750,169.565,43.664,158.244
C03319=1032.517,176.702,393.773,169.562,43.665,158.244
C03320=1032.511,176.454,393.797,169.559,43.666,158.244
C03321=1032.505,176.205,393.820,169.557,43.667,158.244
C03322=1032.499,175.956,393.843,169.553,43.669,158.244
C03323=1032.492,175.708,393.866,169.550,43.670,158.244
C03324=1032.487,175.459,393.889,169.547,43.671,158.244
C03325=1032.480,175.209,393.913,169.544,43.672,158.244
C03326=1032.475,174.960,393.936,169.540,43.674,158.244
C03327=1032.469,174.712,393.959,169.538,43.675,158.244
C03328=1032.462,174.463,393.982,169.535,43.677,158.244
C03329=1032.456,174.214,394.005,169.532,43.678,158.244
C03330=1032.450,173.965,394.028,169.528,43.679,158.244
C03331=1032.444,173.716,394.051,169.526,43.680,158.244
C03332=1032.438,173.468,394.074,169.523,43.682,158.244
C03333=1032.432,173.219,394.097,169.520,43.683,158.244
C03334=1032.426,172.934,394.123,169.516,43.685,158.244
C03335=1032.418,172.651,394.150,169.512,43.686,158.244
C03336=1032.411,172.366,394.176,169.510,43.688,158.244
C03337=1032.404,172.081,394.203,169.506,43.689,158.244
C03338=1032.398,171.833,394.225,169.503,43.691,158.244
C03339=1032.392,171.584,394.248,169.500,43.692,158.244
C03340=1032.386,171.336,394.272,169.498,43.693,158.244
C03341=1032.381,171.087,394.294,169.494,43.695,158.244
C03342=1032.374,170.838,394.317,169.491,43.696,158.244
C03343=1032.368,170.589,394.340,169.488,43.697,158.244
C03344=1032.362,170.340,394.363,169.485,43.698,158.244
C03345=1032.356,170.091,394.386,169.483,43.700,158.244
C03346=1032.351,169.842,394.409,169.479,43.701,158.244
C03347=1032.344,169.593,394.431,169.476,43.703,158.244
C03348=1032.338,169.344,394.454,169.473,43.704,158.244
C03349=1032.333,169.095,394.477,169.470,43.705,158.244
C03350=1032.327,168.847,394.500,169.467,43.706,158.244
C03351=1032.321,168.598,394.523,169.465,43.708,158.244
C03352=1032.315,168.349,394.545,169.461,43.709,158.244
C03353=1032.308,168.099,394.569,169.458,43.711,158.244
C03354=1032.303,167.851,394.592,169.455,43.712,158.244
C03355=1032.297,167.602,394.615,169.453,43.713,158.244
C03356=1032.290,167.353,394.637,169.450,43.714,158.244
C03357=1032.285,167.104,394.660,169.447,43.716,158.245
C03358=1032.279,166.855,394.683,169.444,43.717,158.245
C03359=1032.273,166.606,394.706,169.440,43.719,158.245
C03360=1032.267,166.358,394.728,169.438,43.720,158.245
C03361=1032.261,166.109,394.751,169.435,43.721,158.245
C03362=1032.255,165.860,394.774,169.432,43.723,158.245
C03363=1032.250,165.611,394.797,169.429,43.724,158.245
C03364=1032.243,165.362,394.819,169.426,43.725,158.245
C03365=1032.237,165.114,394.842,169.424,43.726,158.245
C03366=1032.232,164.864,394.865,169.421,43.728,158.245
C03367=1032.226,164.615,394.887,169.418,43.729,158.245
C03368=1032.220,164.366,394.910,169.414,43.731,158.245
C03369=1032.214,164.118,394.933,169.411,43.732,158.245
C03370=1032.208,163.869,394.956,169.409,43.733,158.245
C03371=1032.203,163.620,394.979,169.406,43.734,158.245
C03372=1032.197,163.371,395.002,169.403,43.736,158.245
C03373=1032.191,163.122,395.023,169.400,43.737,158.245
C03374=1032.185,162.873,395.046,169.398,43.739,158.245
C03375=1032.179,162.624,395.069,169.395,43.740,158.245
C03376=1032.173,162.375,395.092,169.392,43.741,158.245
C03377=1032.167,162.127,395.114,169.389,43.742,158.245
C03378=1032.162,161.877,395.137,169.387,43.744,158.245
C03379=1032.156,161.628,395.160,169.384,43.745,158.245
C03380=1032.150,161.380,395.182,169.381,43.746,158.245
C03381=1032.144,161.131,395.205,169.378,43.748,158.245
C03382=1032.139,160.882,395.227,169.374,43.749,158.245
C03383=1032.133,160.633,395.250,169.371,43.750,158.245
C03384=1032.127,160.384,395.272,169.369,43.752,158.245
C03385=1032.121,160.135,395.295,169.366,43.753,158.245
C03386=1032.115,159.886,395.317,169.363,43.755,158.245
C03387=1032.110,159.637,395.340,169.360,43.756,158.245
C03388=1032.104,159.388,395.362,169.358,43.757,158.245
C03389=1032.097,159.139,395.384,169.355,43.759,158.245
C03390=1032.091,158.891,395.407,169.352,43.760,158.245
C03391=1032.085,158.641,395.429,169.349,43.762,158.246
C03392=1032.079,158.393,395.451,169.347,43.763,158.246
C03393=1032.073,158.143,395.473,169.344,43.764,158.246
C03394=1032.067,157.895,395.495,169.341,43.766,158.246
C03395=1032.061,157.646,395.517,169.337,43.768,158.246
C03396=1032.055,157.397,395.539,169.335,43.770,158.246
C03397=1032.049,157.148,395.562,169.332,43.771,158.246
C03398=1032.042,156.864,395.587,169.329,43.773,158.246
C03399=1032.035,156.579,395.612,169.326,43.774,158.246
C03400=1032.028,156.294,395.637,169.323,43.776,158.246
C03401=1032.022,156.009,395.662,169.319,43.777,158.246
C03402=1032.015,155.761,395.685,169.317,43.779,158.246
C03403=1032.010,155.511,395.707,169.314,43.780,158.246
C03404=1032.003,155.262,395.729,169.311,43.782,158.246
C03405=1031.997,155.013,395.751,169.308,43.783,158.246
C03406=1031.991,154.764,395.772,169.305,43.785,158.246
C03407=1031.986,154.516,395.795,169.303,43.787,158.246
C03408=1031.980,154.267,395.817,169.300,43.788,158.246
C03409=1031.973,154.018,395.839,169.297,43.790,158.247
C03410=1031.968,153.768,395.861,169.295,43.791,158.247
C03411=1031.962,153.519,395.883,169.292,43.792,158.247
C03412=1031.955,153.271,395.905,169.289,43.794,158.247
C03413=1031.949,153.021,395.927,169.285,43.795,158.247
C03414=1031.943,152.773,395.948,169.283,43.797,158.247
C03415=1031.937,152.524,395.970,169.280,43.798,158.247
C03416=1031.931,152.275,395.992,169.277,43.800,158.247
C03417=1031.925,152.026,396.014,169.274,43.801,158.247
C03418=1031.919,151.776,396.036,169.272,43.803,158.247
C03419=1031.913,151.527,396.058,169.269,43.805,158.247
C03420=1031.907,151.279,396.080,169.266,43.806,158.247
C03421=1031.901,151.030,396.101,169.264,43.808,158.247
C03422=1031.895,150.781,396.123,169.261,43.810,158.248
C03423=1031.889,150.532,396.145,169.258,43.811,158.248
C03424=1031.883,150.283,396.167,169.256,43.813,158.248
C03425=1031.877,150.034,396.189,169.253,43.814,158.248
C03426=1031.871,149.785,396.210,169.250,43.816,158.248
C03427=1031.865,149.536,396.232,169.247,43.817,158.248
C03428=1031.859,149.287,396.254,169.245,43.818,158.248
C03429=1031.853,149.038,396.275,169.242,43.820,158.248
C03430=1031.847,148.790,396.297,169.239,43.821,158.248
C03431=1031.841,148.540,396.319,169.237,43.823,158.248
C03432=1031.835,148.291,396.341,169.234,43.824,158.248
C03433=1031.829,148.042,396.363,169.231,43.826,158.248
C03434=1031.824,147.793,396.384,169.228,43.827,158.248
C03435=1031.817,147.544,396.406,169.226,43.829,158.248
C03436=1031.811,147.295,396.427,169.223,43.831,158.248
C03437=1031.805,147.046,396.449,169.220,43.832,158.249
C03438=1031.800,146.797,396.470,169.218,43.834,158.249
C03439=1031.793,146.548,396.492,169.215,43.835,158.249
C03440=1031.787,146.299,396.513,169.212,43.837,158.249
C03441=1031.781,146.049,396.535,169.209,43.839,158.249
C03442=1031.775,145.801,396.556,169.207,43.840,158.249
C03443=1031.769,145.552,396.577,169.204,43.842,158.249
C03444=1031.762,145.303,396.599,169.201,43.844,158.249
C03445=1031.756,145.054,396.621,169.199,43.845,158.249
C03446=1031.751,144.805,396.642,169.196,43.847,158.249
C03447=1031.745,144.556,396.664,169.193,43.849,158.249
C03448=1031.738,144.307,396.685,169.191,43.850,158.249
C03449=1031.733,144.058,396.707,169.188,43.852,158.250
C03450=1031.727,143.809,396.728,169.185,43.854,158.250
C03451=1031.720,143.560,396.749,169.183,43.855,158.250
C03452=1031.714,143.312,396.770,169.180,43.857,158.250
C03453=1031.708,143.062,396.792,169.177,43.858,158.250
C03454=1031.702,142.813,396.814,169.175,43.860,158.250
C03455=1031.696,142.563,396.835,169.172,43.862,158.250
C03456=1031.690,142.315,396.856,169.169,43.863,158.250
C03457=1031.684,142.066,396.878,169.167,43.865,158.250
C03458=1031.677,141.817,396.899,169.164,43.866,158.250
C03459=1031.672,141.568,396.920,169.161,43.868,158.250
C03460=1031.666,141.319,396.941,169.158,43.869,158.250
C03461=1031.660,141.071,396.963,169.156,43.871,158.251
C03462=1031.653,140.785,396.986,169.152,43.873,158.251
C03463=1031.647,140.500,397.011,169.149,43.875,158.251
C03464=1031.639,140.215,397.036,169.147,43.876,158.251
C03465=1031.633,139.930,397.060,169.143,43.878,158.251
C03466=1031.626,139.681,397.081,169.140,43.880,158.251
C03467=1031.620,139.432,397.102,169.138,43.881,158.251
C03468=1031.614,139.183,397.124,169.135,43.883,158.251
C03469=1031.609,138.934,397.144,169.132,43.885,158.251
C03470=1031.603,138.685,397.166,169.130,43.886,158.251
C03471=1031.596,138.436,397.187,169.128,43.888,158.252
C03472=1031.590,138.187,397.208,169.125,43.890,158.252
C03473=1031.585,137.938,397.229,169.123,43.891,158.252
C03474=1031.578,137.689,397.250,169.120,43.893,158.252
C03475=1031.572,137.440,397.272,169.117,43.895,158.252
C03476=1031.566,137.190,397.293,169.115,43.896,158.252
C03477=1031.561,136.942,397.314,169.112,43.898,158.252
C03478=1031.554,136.693,397.335,169.109,43.900,158.252
C03479=1031.549,136.444,397.355,169.107,43.901,158.252
C03480=1031.542,136.195,397.377,169.104,43.903,158.252
C03481=1031.536,135.945,397.397,169.101,43.905,158.253
C03482=1031.530,135.697,397.419,169.099,43.906,158.253
C03483=1031.523,135.448,397.440,169.096,43.908,158.253
C03484=1031.518,135.199,397.460,169.093,43.910,158.253
C03485=1031.512,134.949,397.482,169.091,43.911,158.253
C03486=1031.506,134.701,397.502,169.088,43.913,158.253
C03487=1031.500,134.451,397.524,169.085,43.915,158.253
C03488=1031.493,134.202,397.544,169.082,43.916,158.253
C03489=1031.488,133.953,397.565,169.080,43.918,158.253
C03490=1031.482,133.703,397.586,169.077,43.920,158.254
C03491=1031.475,133.455,397.607,169.075,43.922,158.254
C03492=1031.470,133.205,397.628,169.073,43.923,158.254
C03493=1031.463,132.957,397.648,169.070,43.925,158.254
C03494=1031.457,132.707,397.669,169.068,43.926,158.254
C03495=1031.452,132.459,397.690,169.065,43.928,158.254
C03496=1031.445,132.209,397.711,169.062,43.930,158.254
C03497=1031.440,131.961,397.732,169.060,43.931,158.254
C03498=1031.433,131.711,397.752,169.057,43.933,158.254
C03499=1031.428,131.463,397.774,169.054,43.935,158.254
C03500=1031.421,131.213,397.794,169.052,43.936,158.255
C03501=1031.415,130.965,397.815,169.049,43.938,158.255
C03502=1031.410,130.715,397.836,169.046,43.940,158.255
C03503=1031.404,130.466,397.856,169.044,43.941,158.255
C03504=1031.397,130.217,397.877,169.041,43.943,158.255
C03505=1031.391,129.968,397.898,169.038,43.945,158.255
C03506=1031.385,129.719,397.918,169.037,43.946,158.255
C03507=1031.378,129.471,397.939,169.034,43.948,158.255
C03508=1031.372,129.221,397.959,169.031,43.950,158.255
C03509=1031.366,128.971,397.980,169.029,43.952,158.256
C03510=1031.360,128.723,398.001,169.026,43.954,158.256
C03511=1031.353,128.473,398.021,169.024,43.956,158.256
C03512=1031.347,128.225,398.041,169.021,43.957,158.256
C03513=1031.342,127.976,398.061,169.018,43.959,158.256
C03514=1031.335,127.727,398.083,169.016,43.961,158.256
C03515=1031.329,127.478,398.102,169.013,43.963,158.256
C03516=1031.323,127.228,398.123,169.010,43.964,158.256
C03517=1031.317,126.979,398.143,169.008,43.966,158.257
C03518=1031.311,126.730,398.164,169.005,43.968,158.257
C03519=1031.304,126.481,398.184,169.002,43.969,158.257
C03520=1031.298,126.232,398.205,169.000,43.971,158.257
C03521=1031.292,125.983,398.225,168.997,43.973,158.257
C03522=1031.286,125.733,398.246,168.995,43.975,158.257
C03523=1031.280,125.484,398.266,168.993,43.977,158.257
C03524=1031.274,125.235,398.287,168.990,43.978,158.257
C03525=1031.268,124.986,398.307,168.988,43.980,158.258
C03526=1031.261,124.701,398.331,168.984,43.982,158.258
C03527=1031.253,124.417,398.353,168.981,43.984,158.258
C03528=1031.247,124.131,398.376,168.979,43.986,158.258
C03529=1031.240,123.845,398.400,168.975,43.989,158.258
C03530=1031.233,123.597,398.421,168.973,43.990,158.258
C03531=1031.227,123.348,398.441,168.971,43.991,158.258
C03532=1031.221,123.099,398.461,168.968,43.993,158.258
C03533=1031.216,122.850,398.482,168.966,43.995,158.259
C03534=1031.209,122.600,398.502,168.963,43.997,158.259
C03535=1031.203,122.351,398.522,168.960,43.998,158.259
C03536=1031.197,122.103,398.542,168.958,44.000,158.259
C03537=1031.191,121.853,398.563,168.955,44.002,158.259
C03538=1031.185,121.604,398.583,168.953,44.004,158.259
C03539=1031.179,121.355,398.603,168.950,44.006,158.259
C03540=1031.173,121.106,398.623,168.948,44.007,158.259
C03541=1031.167,120.856,398.644,168.946,44.009,158.260
C03542=1031.161,120.608,398.664,168.943,44.011,158.260
C03543=1031.155,120.358,398.684,168.940,44.013,158.260
C03544=1031.149,120.109,398.704,168.938,44.015,158.260
C03545=1031.143,119.860,398.724,168.935,44.016,158.260
C03546=1031.137,119.611,398.745,168.932,44.018,158.260
C03547=1031.131,119.362,398.765,168.931,44.019,158.260
C03548=1031.125,119.113,398.785,168.928,44.021,158.260
C03549=1031.118,118.864,398.805,168.925,44.022,158.260
C03550=1031.113,118.614,398.825,168.923,44.024,158.261
C03551=1031.107,118.366,398.845,168.920,44.026,158.261
C03552=1031.100,118.116,398.866,168.918,44.028,158.261
C03553=1031.094,117.867,398.886,168.915,44.030,158.261
C03554=1031.088,117.618,398.906,168.913,44.031,158.261
C03555=1031.083,117.369,398.926,168.911,44.033,158.261
C03556=1031.077,117.120,398.947,168.908,44.035,158.261
C03557=1031.071,116.871,398.967,168.905,44.037,158.261
C03558=1031.065,116.622,398.986,168.903,44.038,158.261
C03559=1031.058,116.373,399.007,168.900,44.040,158.262
C03560=1031.053,116.124,399.027,168.899,44.042,158.262
C03561=1031.047,115.875,399.047,168.896,44.044,158.262
C03562=1031.041,115.626,399.067,168.893,44.045,158.262
C03563=1031.035,115.376,399.087,168.890,44.047,158.262
C03564=1031.029,115.127,399.107,168.888,44.049,158.262
C03565=1031.023,114.878,399.127,168.885,44.050,158.262
C03566=1031.017,114.629,399.147,168.883,44.052,158.262
C03567=1031.011,114.380,399.167,168.881,44.053,158.262
C03568=1031.005,114.131,399.188,168.878,44.055,158.263
C03569=1030.999,113.882,399.208,168.876,44.057,158.263
C03570=1030.994,113.632,399.227,168.873,44.058,158.263
C03571=1030.988,113.383,399.247,168.871,44.060,158.263
C03572=1030.981,113.134,399.268,168.869,44.062,158.263
C03573=1030.975,112.885,399.288,168.866,44.064,158.263
C03574=1030.969,112.636,399.307,168.864,44.066,158.263
C03575=1030.963,112.387,399.327,168.861,44.067,158.263
C03576=1030.957,112.137,399.347,168.858,44.069,158.264
C03577=1030.951,111.888,399.366,168.857,44.071,158.264
C03578=1030.945,111.639,399.386,168.854,44.073,158.264
C03579=1030.939,111.390,399.406,168.851,44.074,158.264
C03580=1030.934,111.141,399.426,168.849,44.076,158.264
C03581=1030.927,110.891,399.446,168.846,44.078,158.264
C03582=1030.921,110.642,399.466,168.844,44.080,158.264
C03583=1030.915,110.393,399.485,168.841,44.081,158.264
C03584=1030.909,110.144,399.504,168.839,44.083,158.265
C03585=1030.902,109.895,399.525,168.837,44.085,158.265
C03586=1030.896,109.646,399.544,168.834,44.087,158.265
C03587=1030.890,109.397,399.564,168.831,44.089,158.265
C03588=1030.884,109.148,399.583,168.829,44.091,158.265
C03589=1030.878,108.899,399.603,168.826,44.093,158.265
C03590=1030.870,108.613,399.625,168.824,44.095,158.265
C03591=1030.864,108.328,399.648,168.821,44.097,158.266
C03592=1030.857,108.042,399.670,168.818,44.099,158.266
C03593=1030.850,107.758,399.693,168.815,44.101,158.266
C03594=1030.844,107.508,399.712,168.812,44.103,158.266
C03595=1030.837,107.259,399.732,168.811,44.105,158.266
C03596=1030.831,107.010,399.751,168.808,44.107,158.266
C03597=1030.825,106.761,399.771,168.806,44.109,158.267
C03598=1030.819,106.511,399.790,168.803,44.110,158.267
C03599=1030.813,106.263,399.809,168.800,44.112,158.267
C03600=1030.807,106.013,399.829,168.798,44.114,158.267
C03601=1030.800,105.764,399.849,168.795,44.115,158.267
C03602=1030.795,105.515,399.868,168.793,44.117,158.267
C03603=1030.788,105.265,399.887,168.791,44.119,158.267
C03604=1030.782,105.017,399.907,168.788,44.121,158.267
C03605=1030.776,104.767,399.926,168.786,44.123,158.268
C03606=1030.770,104.518,399.946,168.783,44.125,158.268
C03607=1030.764,104.269,399.965,168.781,44.127,158.268
C03608=1030.758,104.020,399.985,168.779,44.128,158.268
C03609=1030.752,103.770,400.004,168.776,44.130,158.268
C03610=1030.745,103.521,400.023,168.774,44.132,158.268
C03611=1030.739,103.272,400.043,168.771,44.134,158.268
C03612=1030.734,103.023,400.062,168.768,44.135,158.268
C03613=1030.728,102.774,400.082,168.767,44.137,158.269
C03614=1030.721,102.525,400.101,168.764,44.139,158.269
C03615=1030.716,102.276,400.120,168.762,44.141,158.269
C03616=1030.710,102.027,400.140,168.759,44.143,158.269
C03617=1030.704,101.777,400.159,168.756,44.145,158.269
C03618=1030.697,101.528,400.178,168.755,44.146,158.269
C03619=1030.691,101.279,400.198,168.752,44.148,158.269
C03620=1030.686,101.030,400.217,168.749,44.150,158.269
C03621=1030.679,100.781,400.236,168.747,44.151,158.270
C03622=1030.673,100.531,400.256,168.744,44.153,158.270
C03623=1030.667,100.282,400.275,168.743,44.155,158.270
C03624=1030.661,100.032,400.294,168.740,44.157,158.270
C03625=1030.655,99.784,400.314,168.737,44.159,158.270
C03626=1030.649,99.534,400.333,168.735,44.161,158.270
C03627=1030.643,99.285,400.352,168.732,44.163,158.270
C03628=1030.637,99.036,400.371,168.730,44.165,158.271
C03629=1030.630,98.787,400.390,168.728,44.166,158.271
C03630=1030.625,98.537,400.409,168.726,44.168,158.271
C03631=1030.618,98.289,400.428,168.723,44.170,158.271
C03632=1030.612,98.040,400.447,168.720,44.172,158.271
C03633=1030.606,97.790,400.466,168.718,44.174,158.271
C03634=1030.599,97.541,400.485,168.715,44.176,158.271
C03635=1030.594,97.292,400.504,168.714,44.178,158.272
